// TwinCAT 3 PLC project Area2
// ProgramVersion: 3.1.4023.0
// libraries:
//   Tc2_DataExchange, * (Beckhoff Automation GmbH)
//   Tc2_MC2, * (Beckhoff Automation GmbH)
//   Tc2_Standard, * (Beckhoff Automation GmbH)
//   Tc2_System, * (Beckhoff Automation GmbH)
//   Tc2_TcpIp, * (Beckhoff Automation GmbH)
//   Tc2_Utilities, * (Beckhoff Automation GmbH)
//   Tc3_BA_Common, * (Beckhoff Automation GmbH)
//   Tc3_Database, * (Beckhoff Automation GmbH)
//   Tc3_JsonXml, * (Beckhoff Automation GmbH)
//   Tc3_Module, * (Beckhoff Automation GmbH)
// project tree:
//   COMMs_ADS/PROTOTYPE/ AdsClient_1.TcPOU (not stored), AdsHandle_1.TcPOU (not stored)
//   COMMs_ADS/Tasks/ AdsHandle.TcPOU, AdsClient.TcPOU (not stored)
//   COMMs_TCP/Types/ DUT.TcDUT (not stored), TcpData.TcDUT (not stored), TcpDataQueue.TcPOU
//   COMMs_TCP/Tasks/ TcpServer1Vision.TcPOU (not stored)
//   DUTs/Enums/ InsertionDirection.TcDUT (not stored), SectionEnum.TcDUT, Homing.TcDUT, SectionStatus.TcDUT, ConveyorMode.TcDUT (not stored), Cover.TcDUT (not stored), EventsEnum.TcTLEO (not stored), MaterialEnums.TcDUT (not stored), MaterialType.TcDUT (not stored), Surface.TcDUT
//   DUTs/Enums/Materials/ Cardboard.TcDUT (not stored), Chipboard.TcDUT (not stored), CornerGuard.TcDUT, WoodBunk.TcDUT (not stored)
//   DUTs/Enums/Robot Tasks/ A22.TcDUT, A21.TcDUT
//   DUTs/Hardware/ A21ToolStorage.TcDUT (not stored), FoldingMachine.TcDUT, Conveyor.TcPOU
//   DUTs/Hardware/Big Machines/ Robot.TcPOU, StrapMachine.TcPOU, WrapMachine.TcPOU
//   DUTs/Hardware/Insertion/Combinations/ ClampInsertion.TcPOU, PneumaticInsertion.TcPOU
//   DUTs/Hardware/Insertion/Drives/ AirPiston.TcPOU, ServoNC.TcPOU, TeknicEIP.TcPOU
//   DUTs/Hardware/Insertion/ Insertion.TcPOU, I_Insertion2D.TcIO
//   DUTs/Hardware/Material Storage/ MaterialStorage.TcPOU, WoodBunkTable.TcPOU
//   DUTs/ ONE_BIT.TcDUT, SuctionPad.TcDUT, VisionFrame.TcDUT (not stored), VisionSuite.TcDUT (not stored)
//   COMMs_ADS/Types/ AdsSocket.TcPOU (not stored), AdsDataQueue.TcPOU, AdsData.TcDUT (not stored)
//   DUTs/Bundle/ Bundle.TcDUT (not stored), CardboardMaterial.TcDUT (not stored), Interval.TcDUT (not stored), Material.TcDUT (not stored), PositionMaterials.TcDUT (not stored)
//   DUTs/Containers/ DynamicQueue.TcPOU, PtrQueue.TcPOU, IntQueue.TcPOU (not stored), Queue.TcPOU (not stored), StringQueue.TcPOU (not stored)
//   EventLogging/ EventLogger.TcIO (not stored), SqlDatabaseAccessor.TcPOU (not stored)
//   / GlobalTextList.TcGTLO (not stored), PlcTask.TcTTO (not stored)
//   GVLs/ GVL.TcGVL, Hardware.TcGVL, MultiProcess.TcGVL
//   POUs/ CallHardware.TcPOU, ConveyorControl.TcPOU, MAIN.TcPOU
//   POUs/Helper Functions/Document/ CreateJsonDocumentManual.TcPOU (not stored), CreateJsonDocumentAuto.TcPOU (not stored), FrameIsValid.TcPOU (not stored), VisionJsonParser.TcPOU
//   POUs/Helper Functions/General/ BufferIsEmpty.TcPOU (not stored), BundleIsValid.TcPOU (not stored), InRange.TcPOU (not stored), PositionIsValid.TcPOU (not stored), TimestructToString.TcPOU (not stored), WithinTolerance.TcPOU
//   POUs/Helper Functions/Material Functions/ GetPositionMasterLength.TcPOU, GetMaterialLength.TcPOU, MatchesMaterialType.TcPOU
//   POUs/Helper Functions/Misc/ ForceSetLifterConveyors.TcPOU, SizeCheck.TcPOU
//   Sections/Concrete/ AreaOutputEx.TcPOU, CardboardCornerGuardEx.TcPOU, ChipboardEx.TcPOU, PaperEx.TcPOU, WoodBunkEx.TcPOU
//   Sections/ I_MaterialSection.TcIO (not stored), SectionEx.TcPOU
// real-time tasks:
//   TASK PlcTask: cycle T#10ms, priority 20, ADS port 350

// ---- DUTs/Enums/Materials/CornerGuard.TcDUT
{attribute 'qualified_only'}
{attribute 'to_string'}
TYPE CornerGuard :
(
	COR48 := 1,
	COR96,
	
	size
);
END_TYPE

// ---- DUTs/Enums/Robot Tasks/A22.TcDUT
{attribute 'qualified_only'}
{attribute 'strict'}
TYPE A22 :
(
	IDLE,
	
	LOAD_CARDBOARD_TOP, //flat cardboards
	LOAD_CARDBOARD_BOTTOM,
	LOAD_CARDBOARD_SIDE,
	REMOVE_CARDBOARD_TOP,
	REMOVE_CARDBOARD_BOTTOM,
	REMOVE_CARDBOARD_SIDE,
	
	TRANSFER_TO_BENDER := 9, //corner cardboards
	TRANSFER_TO_OVERHEAD,
	REMOVE_CARDBOARD_FROM_BENDER,
	LOAD_BENDER_TO_UPPER_CORNER,
	LOAD_BENDER_TO_LOWER_CORNER,
	LOAD_OVERHEAD_TO_UPPER_CORNER,
	LOAD_OVERHEAD_TO_LOWER_CORNER,
	
	REMOVE_CARDBOARD_UPPER_CORNER,
	REMOVE_CARDBOARD_LOWER_CORNER,
	REMOVE_CARDBOARD_OVERHEAD := 18,
	
	LOAD_CORNER_GUARD_UPPER := 20, //corner guards
	LOAD_CORNER_GUARD_LOWER,
	REMOVE_CORNER_GUARD_UPPER,
	REMOVE_CORNER_GUARD_LOWER,
	
	size
);
END_TYPE

// ---- DUTs/Enums/SectionEnum.TcDUT
{attribute 'qualified_only'}
TYPE SectionEnum :
(
	NULL_SECTION := -1,
	PAPER,
	CARDBOARD_CORNERGUARD,
	CHIPBOARD,
	WOOD_BUNK,
	OUTPUT,
	
	size
);
END_TYPE

// ---- DUTs/Hardware/FoldingMachine.TcDUT
TYPE FoldingMachine :
STRUCT
	enable AT %Q* : BOOL;
	foldPos0 AT %Q* : REAL;
	foldPos1 AT %Q* : REAL;
	
	activeMaterial : STRING;
	
	ready AT %I* : BOOL;
	busy AT %I* : BOOL;
	done AT %I* : BOOL;
	error AT %I* : BOOL;
END_STRUCT
END_TYPE

// ---- DUTs/ONE_BIT.TcDUT
TYPE ONE_BIT :
STRUCT
	e1 : BIT;
END_STRUCT
END_TYPE

// ---- DUTs/Enums/Robot Tasks/A21.TcDUT
{attribute 'qualified_only'}
{attribute 'strict'}
TYPE A21 :
(
	IDLE,
	STAGE_BUNK,
	REMOVE_BUNK_FROM_STAGE,
	
	LOAD_BUNK_TO_TOP := 4,
	LOAD_BUNK_TO_SIDE,
	LOAD_BUNK_TO_BOTTOM,
	REMOVE_BUNK_FROM_TOP,
	REMOVE_BUNK_FROM_SIDE,
	REMOVE_BUNK_FROM_BOTTOM,
	
	GET_CHIPBOARD_FROM_SKID := 11,
	REMOVE_CHIPBOARD_FROM_TOOL,
	PLACE_CHIPBOARD_TO_TOP,
	PLACE_CHIPBOARD_TO_BOTTOM,
	REMOVE_CHIPBOARD_TOP,
	REMOVE_CHIPBOARD_BOTTOM,
	
	FIX_CHIPBOARD_ORIENTATION := 19,
	
	//testing only
	MOVE_HOME := 21,
	MOVE_POSITION1,
	MOVE_POSITION2,
	MOVE_UP,
	MOVE_DOWN,
	
	DIRECT_BUNK_TO_TOP := 27,
	DIRECT_BUNK_TO_SIDE,
	DIRECT_BUNK_TO_BOTTOM,
	
	INSPECT_BUNK := 31,
	INSPECT_CHIPBOARD,
	
	TOOL_CHANGE_BUNK := 34,
	TOOL_CHANGE_CHIPBOARD,
	
	size
);
END_TYPE

// ---- DUTs/Enums/Homing.TcDUT
{attribute 'qualified_only'}
{attribute 'strict'}
TYPE Homing :
(
	IDLE,
	HOME_OUT,
	HOME_FINAL,
	STOP,
	SET,
	DONE,
	REDO
);
END_TYPE

// ---- DUTs/Enums/SectionStatus.TcDUT
{attribute 'qualified_only'}
//{attribute 'strict'}
TYPE SectionStatus :
(
	IDLE,
	ALIGNING,
	ACTIVE,
	CLEARING,
	COMPLETE,
	
	size
);
END_TYPE

// ---- DUTs/Enums/Surface.TcDUT
{attribute 'qualified_only'}
//{attribute 'strict'}
TYPE Surface :
(
	TOP,
	LEFT,
	RIGHT,
	BOTTOM,
	
	TOP_LEFT,
	TOP_RIGHT,
	BOTTOM_LEFT,
	BOTTOM_RIGHT,
	
	size
);
END_TYPE

// ---- DUTs/SuctionPad.TcDUT
TYPE SuctionPad :
STRUCT
	enable AT %Q* : BOOL;
	readback AT %I* : BOOL;
END_STRUCT
END_TYPE

// ---- GVLs/GVL.TcGVL
{attribute 'qualified_only'}
VAR_GLOBAL CONSTANT
	maxPairs : USINT := 16;
	initArraySize : USINT := 4;
	maxQueue : INT := 16;
	
	nullPos : REAL := -1;
	
	numMaterials : INT := 32;
	allMaterials : ARRAY[0..numMaterials] OF Material := [
		(code := 'PAP28', width := 28, length := -1),
		
		(code := 'CAR20S', width := 20, length := 30),
		(code := 'CAR20M', width := 20, length := 45),
		(code := 'CAR20L', width := 20, length := 60),
		(code := 'CAR28S', width := 28, length := 30),
		(code := 'CAR28M', width := 28, length := 45),
		(code := 'CAR28L', width := 28, length := 60),
		
		(code := 'COR48', width := 1.5, length := 48),
		(code := 'COR96', width := 1.5, length := 96),
		
		(code := 'CIP18', width := 20, length := 18),
		(code := 'CIP54', width := 20, length := 54),
		
		(code := 'WDT20', width := 20, length := 2.5),
		(code := 'WDT22', width := 22, length := 2.5),
		(code := 'WDT28', width := 28, length := 2.5),
		
		(code := 'WDB20', width := 20, length := 2.5),
		(code := 'WDB22', width := 22, length := 2.5),
		(code := 'WDB28', width := 28, length := 2.5),
		
		(code := 'WDS08', width := 8, length := 2.5),
		(code := 'WDS10', width := 10, length := 2.5),
		(code := 'WDS12', width := 12, length := 2.5),
		(code := 'WDS14', width := 14, length := 2.5),
		(code := 'WDS8x8', width := 16, length := 2.5),
		(code := 'WDS8x10', width := 18, length := 2.5),
		(code := 'WDS20', width := 20, length := 2.5),
		(code := 'WDS22', width := 22, length := 2.5),
		(code := 'WDS12x12', width := 24, length := 2.5),
		(code := 'WDS12x14', width := 26, length := 2.5),
		(code := 'WDS28', width := 28, length := 2.5),
		(code := 'WDS20x10', width := 30, length := 2.5),
		(code := 'WDS20x12', width := 32, length := 2.5),
		
		(code := 'WDW20', width := 20, length := 6),
		(code := 'WDW22', width := 22, length := 6)]; //+1 null material

	nullBundle : Bundle;
	
	conveyorLength : REAL := 0;
	precisionTolerance : REAL := 0.05 * 25.4;
END_VAR
VAR_GLOBAL
	bundleOut : Bundle;
END_VAR

// ---- GVLs/Hardware.TcGVL
//{attribute 'qualified_only'}
VAR_GLOBAL CONSTANT
	numConveyors : INT := 20;
END_VAR
VAR_GLOBAL
	allConveyors : ARRAY[0..numConveyors] OF Conveyor;

	robots : ARRAY[1..6] OF Robot;
	
	(*
	names for moving parts should be in the following format: <type> <location> <left/right>
	*)
	
	//A23 - PAPER
	(*
	wrapperPaper : WrapMachine;
	*)
	//new
	wrapperA23 : WrapMachine;
	//-------------
	
	//A22 - CARDBOARD + CORNER GUARD
	(*
	cardboardSkid : ARRAY[Surface.LEFT..Surface.RIGHT] OF MaterialStorage;
	cornerGuardMagazine : ARRAY[Surface.LEFT..Surface.RIGHT] OF MaterialStorage;
	
	cardboardBender : ARRAY[Surface.LEFT..Surface.RIGHT] OF FoldingMachine;
	insertionCardboardCornerGuardSides : ARRAY[Surface.LEFT..Surface.RIGHT] OF ClampInsertion;
	insertionCardboardCornerGuardBottom : TeknicEIP;
	
	wrapperCardboardCornerguard : WrapMachine;
	*)
	//new
	cardboardBenderLeft, cardboardBenderRight : FoldingMachine;
	
	cardboardSkidLeft, cardboardSkidRight : MaterialStorage;
	cornerGuardMagazineLeft, cornerGuardMagazineRight : MaterialStorage;
	insertionA22Left, insertionA22Right : ClampInsertion;
	insertionA22Bottom : TeknicEIP;
	
	wrapperA22 : WrapMachine;
	overhead : STRING;
	//-------------
	
	
	//A21 - CHIPBOARD + WOOD BUNK
	(*
	toolStorage : ARRAY[Surface.LEFT..Surface.RIGHT] OF A21ToolStorage;
	
	chipboardSkid : ARRAY[Surface.LEFT..Surface.RIGHT] OF MaterialStorage;
	
	woodBunkMagazine : ARRAY[Surface.LEFT..Surface.RIGHT] OF MaterialStorage;
	stagingTable : ARRAY[Surface.LEFT..Surface.RIGHT] OF WoodBunkTable;
	strapper : StrapMachine;
	insertionWoodBunkSides : ARRAY[Surface.LEFT..Surface.RIGHT] OF PneumaticInsertion;
	insertionWoodBunkBottom : TeknicEIP;
	*)
	//new
	toolStorageA21Left, toolStorageA21Right : A21ToolStorage;
	
	chipboardSkidLeft, chipboardSkidRight : MaterialStorage;
	woodBunkMagazineLeft, woodBunkMagazineRight : MaterialStorage;
	
	stagingTableLeft, stagingTableRight : WoodBunkTable;
	strapperA21 : StrapMachine;
	
	insertionA21Left, insertionA21Right : PneumaticInsertion;	
	insertionA21Bottom : TeknicEIP;
	//-------------
	
	//A25 - OUTPUT
END_VAR

// ---- GVLs/MultiProcess.TcGVL
//{attribute 'qualified_only'}
VAR_GLOBAL
	iecCriticalSection : FB_IecCriticalSection; //must be used if communication routines are separated into their own core/task
END_VAR

// ---- DUTs/Hardware/Insertion/I_Insertion2D.TcIO
INTERFACE I_Insertion2D

METHOD ABSTRACT align : BOOL
VAR_INPUT
	targetPos : REAL;
END_VAR
END_METHOD

PROPERTY Busy : BOOL
GET
END_GET
SET
END_SET
END_PROPERTY

PROPERTY Contact : BOOL
GET
END_GET
SET
END_SET
END_PROPERTY

PROPERTY Home : BOOL
GET
END_GET
SET
END_SET
END_PROPERTY

METHOD ABSTRACT homingSequence : BOOL
VAR_INPUT
END_VAR
END_METHOD

METHOD ABSTRACT press : BOOL
VAR_INPUT
END_VAR
END_METHOD

METHOD ABSTRACT release : BOOL
VAR_INPUT
END_VAR
END_METHOD

PROPERTY ScrewPos : LREAL
GET
END_GET
SET
END_SET
END_PROPERTY

PROPERTY SliderPos : LREAL
GET
END_GET
SET
END_SET
END_PROPERTY

METHOD ABSTRACT traverse : BOOL
VAR_INPUT
	direction : MC_Direction;
END_VAR
END_METHOD

END_INTERFACE

// ---- DUTs/Hardware/Conveyor.TcPOU
FUNCTION_BLOCK Conveyor
VAR_OUTPUT
	operation : ConveyorMode;
	request : ConveyorMode;
	
	enable AT %Q* : BOOL := TRUE;
	direction AT %Q* : BOOL; //FALSE = forward, TRUE = backward
	pulse AT %Q* : BOOL;
	reset AT %Q* : BOOL;
	
	error AT %I* : BOOL;
	sensorEntry AT %I* : BOOL;
	sensorExit AT %I* : BOOL;
	
	//vertical conveyors only
	requestLifter: BOOL;

	lifterEnable AT %Q* : BOOL := TRUE;
	lifterDirection AT %Q* : BOOL; //FALSE = up, TRUE = down
	lifterPulse AT %Q* : BOOL;
	lifterReset AT %Q* : BOOL;
	
	lifterError AT %I* : BOOL;
	extended AT %I* : BOOL;
	retracted AT %I* : BOOL;
END_VAR
VAR_OUTPUT
	position AT %I* : REAL;
	velocity AT %I* : REAL;
END_VAR
VAR
	hasLifter : BOOL;
	
	//pulses are assumed to be low-high-low
	pulser : TP;
	lifterPulser : TP;
END_VAR
VAR_STAT CONSTANT
	pulseWidth : TIME := T#25MS;
END_VAR

pulser(IN:= , PT:= pulseWidth, Q=> pulse, ET=> );

direction := (operation = ConveyorMode.BACKWARD);

pulser.IN := 
	enable AND 
	NOT error AND 
	NOT reset AND 
	(operation = ConveyorMode.FORWARD OR operation = ConveyorMode.BACKWARD);

IF pulser.IN AND NOT pulser.Q THEN
	pulser.IN := FALSE;
END_IF

lifterPulser(IN:= , PT:= pulseWidth, Q=> lifterPulse, ET=> );

lifterPulser.IN := 
	hasLifter AND
	lifterEnable AND 
	NOT lifterError AND 
	NOT lifterReset AND 
	requestLifter;
	
IF lifterPulser.IN AND NOT lifterPulser.Q THEN
	lifterPulser.IN := FALSE;
END_IF

METHOD backward : BOOL
VAR_INPUT
END_VAR
END_METHOD

METHOD extend : BOOL
VAR_INPUT
END_VAR
END_METHOD

METHOD forward : BOOL
VAR_INPUT
END_VAR
END_METHOD

METHOD occupied : BOOL
occupied := sensorExit OR sensorEntry;
END_METHOD

METHOD reset : BOOL
VAR_INPUT
END_VAR
position := 0;
velocity := velocity; //no change

extend();
END_METHOD

METHOD retract : BOOL
VAR_INPUT
END_VAR
END_METHOD

METHOD setOperation : BOOL
VAR_INPUT
	newOperation : ConveyorMode;
END_VAR
operation := newOperation;
END_METHOD

METHOD setRequest : BOOL
VAR_INPUT
	requestedMode : ConveyorMode;
END_VAR
request := requestedMode;
END_METHOD

METHOD target : BOOL
VAR_INPUT
	targetPosition : REAL;
END_VAR
END_METHOD

END_FUNCTION_BLOCK

// ---- DUTs/Hardware/Big Machines/Robot.TcPOU
FUNCTION_BLOCK Robot
VAR_OUTPUT
	forceStop AT %Q* : BOOL;
	resetSignal AT %Q* : BOOL;
	
	taskID AT %Q* : INT;
	parameters AT %Q* : ARRAY[1..3] OF INT;
	
	outputs AT %Q* : ARRAY[1..50] OF INT;
	inputs AT %I* : ARRAY[1..20] OF INT;
	
	completedTask AT %I* : INT;
	tool AT %I* : SectionEnum;
	
	reserved : BOOL;
	reservation : SectionEnum := SectionEnum.NULL_SECTION;
	
	operational : BOOL;
	ready : BOOL;
	//busy : BOOL;
	done : BOOL;
	error : BOOL;
	errId : DINT;
END_VAR
VAR
	step : (SEND_COMMAND, WAIT);
END_VAR
VAR_STAT CONSTANT	
	emptyRegister : ARRAY[0..2] OF INT := [3(0)];
END_VAR

IF completedTask = taskID THEN
	done := TRUE;
END_IF

METHOD command : BOOL
VAR_INPUT
	task : INT;
	param1 : INT;
	param2 : INT;
	param3 : INT;
END_VAR
//command := reserve();

//IF command THEN
	(*
	taskId := task;
	parameters[1] := param1;
	parameters[2] := param2;
	parameters[3] := param3;
	*)
	
	outputs[1] := task;
	outputs[2] := param1;
	outputs[3] := param2;
	outputs[4] := param3;
//END_IF
END_METHOD

METHOD eStop : BOOL
VAR_INPUT
END_VAR
forceStop := TRUE;
eStop := TRUE;
END_METHOD

METHOD release : BOOL
VAR_INPUT
	sectionReservation : SectionEnum;
END_VAR
IF reservation = sectionReservation AND reserved THEN
	reservation := -1;
	reserved := FALSE;
	release := TRUE;
END_IF
END_METHOD

METHOD reserve : BOOL
VAR_INPUT
	sectionReservation : SectionEnum;
END_VAR
(*
some sections may use the same robot so it must be reserved before use
both sections need to check if the robot is open to commands before use
*)
IF
	(reserved AND reservation = SectionReservation) OR_ELSE
	(NOT reserved OR sectionReservation = SectionEnum.NULL_SECTION)
THEN
	reservation := sectionReservation;
	reserved := TRUE;
	reserve := TRUE;
END_IF
END_METHOD

METHOD reset : BOOL
release(reservation);

resetSignal := TRUE;
done := FALSE;
taskID := 0;
parameters := emptyRegister;

MEMSET(ADR(outputs), 0, SIZEOF(outputs));

IF ready AND completedTask = 0 THEN
	resetSignal := FALSE;
	reset := TRUE;
END_IF
END_METHOD

METHOD resume : BOOL
VAR_INPUT
END_VAR
forceStop := FALSE;

resume := NOT error AND errId = 0;
END_METHOD

METHOD setCommandAndWait : BOOL
VAR_INPUT
	task, param1, param2, param3 : INT;
END_VAR
(*
this method sends a command and waits for completion
MAKE SURE TO RESERVE THE ROBOT FIRST
*)
CASE step OF
	SEND_COMMAND: //send command
		command(
			task:= task, 
			param1:= param1, 
			param2:= param2, 
			param3:= param3);
		
		step := WAIT;
		
	WAIT:
		IF done THEN
			release(reservation);
			
			IF NOT reset() THEN
				RETURN;
			END_IF
			
			step := 0;
			
			setCommandAndWait := TRUE;
		END_IF
END_CASE
END_METHOD

METHOD setParamsAndWait : BOOL
VAR_INPUT
	newOutputs : REFERENCE TO ARRAY[1..50] OF INT;
END_VAR
outputs := newOutputs;

IF done THEN
	//release(); //let each section manually release
	
	IF NOT reset() THEN
		RETURN;
	END_IF
	
	step := 0;

	setParamsAndWait := TRUE;
END_IF
END_METHOD

END_FUNCTION_BLOCK

// ---- DUTs/Hardware/Big Machines/WrapMachine.TcPOU
FUNCTION_BLOCK WrapMachine
VAR_OUTPUT
	error AT %I* : BOOL;
	ready AT %I* : BOOL;
	busy AT %I* : BOOL;
	done (*AT %I**) : BOOL;
	home AT %I* : BOOL;
	
	rotations AT %Q* : INT;
	execute AT %Q* : BOOL;
	enable AT %Q* : BOOL;
	reset AT %Q* : BOOL;
	
	timeout : BOOL;
END_VAR
VAR
	holdPost : TON;
	delay : TON;
	
	start : BOOL;
	step : (SETUP, RUN, WAIT);
END_VAR
VAR_STAT CONSTANT
	pulseTime : TIME := T#100MS;
	holdTime : TIME := T#500MS;
	maxDelay : TIME := T#30S;
END_VAR

holdPost(IN:= , PT:= holdTime, Q=> , ET=> );
delay(IN:= step > 0, PT:= maxDelay, Q=> , ET=> );

IF delay.Q THEN
	delay.IN := FALSE;
	timeout := TRUE;
	busy := FALSE;
	step := SETUP;
END_IF

CASE step OF
	SETUP:
		busy := FALSE;
		IF error THEN
			reset := NOT reset;
			enable := FALSE;//NOT enable;
			
		ELSE
			reset := FALSE;
			enable := TRUE;
			
			IF start THEN
				start := FALSE;
				step := RUN;
			END_IF
			
		END_IF
	
	RUN:
		execute := TRUE;
		IF execute AND NOT home THEN
			execute := FALSE;
			step := WAIT;
		END_IF
		
	WAIT:
		IF home THEN
			holdPost.IN := TRUE;
			enable := FALSE;
			execute := FALSE;
		END_IF
		
		IF holdPost.Q THEN
			holdPost.IN := FALSE;
			done := TRUE;
			step := 0;
		END_IF
		
END_CASE

METHOD clear : BOOL
VAR_INPUT
END_VAR
(*
reset should be continuously called until machine returns evidence that it is ready again
machine is expected to not respond to reset signals if it is already in an idle state
*)
enable := FALSE;
execute := FALSE;

IF error THEN
	reset := NOT reset;
	clear := NOT error;

ELSE
	reset := FALSE;
	clear := TRUE;
	
END_IF
END_METHOD

METHOD wrap : BOOL
VAR_INPUT
	reqRotations : INT;
END_VAR
IF ready AND NOT busy AND NOT error THEN
	rotations := reqRotations;
	busy := TRUE;
	start := TRUE;
	wrap := TRUE;
END_IF
END_METHOD

END_FUNCTION_BLOCK

// ---- DUTs/Hardware/Material Storage/MaterialStorage.TcPOU
FUNCTION_BLOCK MaterialStorage
VAR_OUTPUT
	slots : ARRAY[1..GVL.maxQueue] OF STRING;
	//units : ARRAY[0..GVL.maxQueue] OF INT;
	
	empty AT %I* : ARRAY[1..GVL.maxQueue] OF BOOL;
END_VAR

METHOD findSlot : BOOL
VAR_INPUT
	materialID : STRING;
END_VAR
VAR_OUTPUT
	atSlot : INT := -1;
END_VAR
VAR
	i : INT;
END_VAR
IF materialID = '' THEN
	RETURN;
END_IF

FOR i:=0 TO GVL.maxQueue BY 1 DO
	IF slots[i] = materialID THEN
		atSlot := i;
		findSlot := TRUE;
		RETURN;
	END_IF
END_FOR
END_METHOD

METHOD getSlotsAsArray : POINTER TO STRING
getSlotsAsArray := ADR(slots);
END_METHOD

METHOD setupSlots : BOOL
VAR_INPUT
	setSlots : REFERENCE TO ARRAY[1..GVL.maxQueue] OF STRING;
END_VAR
slots := setSlots;
END_METHOD

END_FUNCTION_BLOCK

// ---- DUTs/Hardware/Insertion/Combinations/ClampInsertion.TcPOU
FUNCTION_BLOCK ClampInsertion EXTENDS Insertion
VAR
	slider : ServoNC;
	screw : TeknicEIP;
END_VAR

slider(
	bEnable:= enable, 
	home=> , 
	outerLimit=> , 
	innerLimit=> , 
	ready=> , 
	busy=> , 
	error=> , 
	homeSet=> , 
	position=> sliderPos);

screw(
	bEnable:= enable, 
	home=> , 
	outerLimit=> , 
	innerLimit=> , 
	done=> , 
	homeSet=> , 
	busy=> , 
	error=> , 
	position=> screwPos);

home := screw.home AND slider.home;
busy := slider.busy OR screw.busy;
error := slider.error OR screw.error;

METHOD align : BOOL
VAR_INPUT
	targetPos : REAL;
END_VAR
align := slider.moveAbsolute(targetPos := targetPos);
END_METHOD

METHOD homingSequence : BOOL
IF NOT slider.homeSet THEN
	slider.homingSequence();
END_IF

IF NOT screw.homeSet THEN
	screw.homingSequence();
END_IF

homingSequence := slider.homeSet AND screw.homeSet;
END_METHOD

METHOD press : BOOL
screw.moveContinuous(direction := MC_Negative_Direction);
END_METHOD

METHOD release : BOOL
VAR_INPUT
END_VAR
screw.moveContinuous(direction := MC_Positive_Direction);
END_METHOD

METHOD traverse : BOOL
VAR_INPUT
	direction : MC_Direction;
END_VAR
slider.moveContinuous(direction := direction);
END_METHOD

END_FUNCTION_BLOCK

// ---- DUTs/Hardware/Insertion/Insertion.TcPOU
FUNCTION_BLOCK ABSTRACT Insertion //IMPLEMENTS I_Insertion2D
VAR_INPUT CONSTANT
	enable : BOOL;
END_VAR
VAR_OUTPUT
	contact AT %I* : BOOL;
	home : BOOL;
	busy : BOOL;
	error : BOOL;
	
	sliderPos : LREAL;
	screwPos : LREAL;
END_VAR
(*
this abstract FB encapsulates 2 drives into a generic insertion machine
this FB cannot be used to instantiate insertions, it can only be used to refer/point to existing insertions
RETURN VALUES FOR THE METHODS ARE MEANINGLESS
*)

METHOD ABSTRACT align : BOOL
VAR_INPUT
	targetPos : REAL;
END_VAR
END_METHOD

METHOD ABSTRACT homingSequence : BOOL
VAR_INPUT
END_VAR
END_METHOD

METHOD ABSTRACT press : BOOL
VAR_INPUT
END_VAR
END_METHOD

METHOD ABSTRACT release : BOOL
VAR_INPUT
END_VAR
END_METHOD

METHOD ABSTRACT traverse : BOOL
VAR_INPUT
	direction : MC_Direction;
END_VAR
END_METHOD

END_FUNCTION_BLOCK

// ---- DUTs/Hardware/Insertion/Drives/ServoNC.TcPOU
FUNCTION_BLOCK ServoNC
VAR_INPUT CONSTANT
	bEnable : BOOL;
END_VAR
VAR_OUTPUT
	home AT %I* : BOOL;
	outerLimit AT %I* : BOOL;
	innerLimit AT %I* : BOOL;
	
	ready : BOOL;
	busy : BOOL;
	error : BOOL;
	homeSet : BOOL;
	
	position : LREAL;
END_VAR
VAR
	axis : AXIS_REF;
	
	mcReadPosition : MC_ReadActualPosition;
	mcReset : MC_Reset;
	
	mcPower : MC_Power;
	mcMoveAbsolute : MC_MoveAbsolute;
	mcMoveRelative : MC_MoveRelative;
	mcMoveVelocity : MC_MoveVelocity;
	
	mcStop : MC_Stop;
	mcSetPosition : MC_SetPosition;
	
	step : Homing;
END_VAR
VAR_STAT CONSTANT
	targetingVelocity : INT := 500;
	continuousVelocity : INT := 200;
END_VAR

mcReadPosition(
	Axis:= axis, 
	Enable:= TRUE, 
	Valid=> , 
	Busy=> , 
	Error=> , 
	ErrorID=> , 
	Position=> position);

mcReset(
	Axis:= axis, 
	Execute:= , 
	Done=> , 
	Busy=> , 
	Error=> , 
	ErrorID=> );

mcPower(
	Axis:= axis, 
	Enable:= bEnable, 
	Enable_Positive:= TRUE, 
	Enable_Negative:= TRUE, 
	Override:= 100, 
	BufferMode:= , 
	Options:= , 
	Status=> , 
	Busy=> , 
	Active=> , 
	Error=> , 
	ErrorID=> );

mcMoveAbsolute(
	Axis:= axis, 
	Execute:= , 
	Position:= , 
	Velocity:= targetingVelocity, 
	Acceleration:= , 
	Deceleration:= , 
	Jerk:= , 
	BufferMode:= , 
	Options:= , 
	Done=> , 
	Busy=> , 
	Active=> , 
	CommandAborted=> , 
	Error=> , 
	ErrorID=> );
		
mcMoveRelative(
	Axis:= axis, 
	Execute:= , 
	Distance:= ,
	Velocity:= targetingVelocity, 
	Acceleration:= , 
	Deceleration:= , 
	Jerk:= , 
	BufferMode:= , 
	Options:= , 
	Done=> , 
	Busy=> , 
	Active=> , 
	CommandAborted=> , 
	Error=> , 
	ErrorID=> );
	
mcMoveVelocity(
	Axis:= axis, 
	Execute:= , 
	Velocity:= continuousVelocity, 
	Acceleration:= , 
	Deceleration:= , 
	Jerk:= , 
	Direction:= , 
	BufferMode:= , 
	Options:= , 
	InVelocity=> , 
	Busy=> , 
	Active=> , 
	CommandAborted=> , 
	Error=> , 
	ErrorID=> );
	
mcStop(
	Axis:= axis, 
	Execute:= , 
	Deceleration:= , 
	Jerk:= , 
	Options:= , 
	Done=> , 
	Busy=> , 
	Active=> , 
	CommandAborted=> , 
	Error=> , 
	ErrorID=> );

mcSetPosition(
	Axis:= axis, 
	Execute:= , 
	Position:= , 
	Mode:= , 
	Options:= , 
	Done=> , 
	Busy=> , 
	Error=> , 
	ErrorID=> );
	
busy := mcMoveAbsolute.Busy OR mcMoveRelative.Busy OR mcMoveVelocity.Busy OR mcSetPosition.Busy OR mcReset.Busy OR mcStop.Busy OR step <> 0;
error := mcMoveAbsolute.Error OR mcMoveRelative.Error OR mcMoveVelocity.Error OR mcSetPosition.Error OR mcReset.Error OR mcStop.Error OR step <> 0;
ready := bEnable AND NOT busy AND homeSet;

IF step <> 0 THEN
	mcReset.Execute := FALSE;
	mcMoveAbsolute.Execute := FALSE;
	mcMoveRelative.Execute := FALSE;
	mcMoveVelocity.Execute := FALSE;
	mcStop.Execute := FALSE;
	mcSetPosition.Execute := FALSE;
END_IF

METHOD homingSequence : BOOL
CASE step OF
	Homing.IDLE:
		IF bEnable THEN
			step := Homing.REDO;
		END_IF
		
	Homing.REDO:
		IF mcMoveVelocity.Execute AND NOT innerLimit THEN
			mcMoveVelocity.Execute := FALSE;
			step := Homing.HOME_OUT;
			RETURN;
		END_IF
		
		mcMoveVelocity.Direction := MC_Negative_Direction;
		mcMoveVelocity.Execute := TRUE;
		
	Homing.HOME_OUT:
		IF mcMoveVelocity.Execute AND NOT home THEN //if reached home
			mcMoveVelocity.Execute := FALSE;
			step := Homing.STOP;
			RETURN;
		END_IF
		
		mcMoveVelocity.Direction := MC_Positive_Direction;
		mcMoveVelocity.Execute := TRUE;
		
	Homing.STOP:
		IF mcStop.Execute AND mcStop.Done THEN
			mcStop.Execute := FALSE;
			step := Homing.SET;
			RETURN;
		END_IF
		
		mcStop.Execute := TRUE;
		
	Homing.SET:
		IF mcSetPosition.Execute AND mcSetPosition.Done THEN
			mcSetPosition.Execute := FALSE;
			homingSequence := TRUE;
			step := Homing.IDLE;
			RETURN;
		END_IF
		
		mcSetPosition.Position := 0;
		mcSetPosition.Execute := TRUE;
		
END_CASE
END_METHOD

METHOD moveAbsolute : BOOL
VAR_INPUT
	targetPos : LREAL;
END_VAR
IF NOT busy AND NOT error THEN
	mcMoveAbsolute.Position := targetPos;
END_IF
moveAbsolute := mcMoveAbsolute.Done;
END_METHOD

METHOD moveContinuous : BOOL
VAR_INPUT
	direction : MC_Direction;
END_VAR
mcMoveVelocity.Direction := direction;

mcMoveVelocity.Execute := TRUE;

moveContinuous := NOT mcMoveVelocity.Error;
END_METHOD

METHOD moveRelative : BOOL
VAR_INPUT
	distance : LREAL;
END_VAR
mcMoveRelative.Distance := distance;

moveRelative := mcMoveRelative.Done;
END_METHOD

METHOD reset : BOOL
VAR_INPUT
END_VAR
mcReset.Execute := TRUE;

reset := mcReset.Done;
END_METHOD

METHOD stop : BOOL
VAR_INPUT
END_VAR
END_METHOD

END_FUNCTION_BLOCK

// ---- DUTs/Hardware/Insertion/Drives/TeknicEIP.TcPOU
FUNCTION_BLOCK TeknicEIP //EXTENDS EncodedDrive
VAR_INPUT CONSTANT
	bEnable : BOOL;
END_VAR
VAR_OUTPUT
	enable AT %Q* : BOOL; //enable + pulses
	A AT %Q* : BOOL; //direction (F = inwards, T = outwards)
	B AT %Q* : BOOL; //home bit
	brakeRelease AT %Q* : BOOL;
	
	contact AT %I* : BOOL;
	
	home AT %I* : BOOL;
	outerLimit AT %I* : BOOL;
	innerLimit AT %I* : BOOL;
	done AT %I* : BOOL;	
	
	homeSet : BOOL;
	busy : BOOL;
	error : BOOL;
	
	position : LREAL;
	targetPos : LREAL;
END_VAR
VAR
	mode : (HOLD, TARGET, CONTINUOUS);
	
	resetTimer : TP;
	pulser : TON;
	requestedPulses : INT;
	
	step : Homing;//(IDLE, HOME_UP, HOME_FINAL, DOWN, REDO_HOME, HOME_DONE);
END_VAR
VAR_STAT CONSTANT
	resetTime : TIME := T#1000MS;
	pulseWidth : TIME := T#25MS;
	unitsPerPulse : INT := 800; //800 Teknic units per revolution
	distancePerPulse : INT := 5; //5mm per revolution
END_VAR

IF NOT bEnable THEN
	RETURN;
END_IF

resetTimer(IN:= , PT:= resetTime, Q=> , ET=> );
IF resetTimer.Q THEN
	brakeRelease := FALSE;
	enable := FALSE;
	RETURN;
END_IF
resetTimer.IN := FALSE;


CASE mode OF
	HOLD:
		//
	
	TARGET:
		IF WithinTolerance(position, target, unitsPerPulse) THEN
			requestedPulses := 0;
			mode := HOLD;
			
		ELSIF position < target THEN
			A := TRUE;
			requestPulses(1);
		ELSIF position > target THEN
			A := FALSE;
			requestPulses(1);
		END_IF

	CONTINUOUS:
		requestPulses(1);
		
END_CASE

IF home OR innerLimit OR outerLimit THEN
	requestedPulses := 0;
	mode := HOLD;
END_IF

sequence();

METHOD homingSequence : BOOL
CASE step OF
	Homing.IDLE:
		enable := FALSE;
		A := FALSE;
		B := FALSE;
		brakeRelease := TRUE;
		
		homeSet := FALSE;
		step := Homing.REDO;
		
	Homing.REDO: //let insertion drop to inner limit before homing
		enable := FALSE;
		A := FALSE;
		B := FALSE;
		brakeRelease := TRUE;
		
		IF NOT innerLimit THEN
			enable := TRUE;
			step := Homing.HOME_OUT;
		END_IF
	
	Homing.HOME_OUT:
		enable := TRUE;
		A := FALSE;
		B := TRUE;
		brakeRelease := TRUE;
		
		IF NOT home THEN
			B := FALSE;
			step := Homing.DONE;
		END_IF
		
	Homing.DONE:
		enable := TRUE;
		A := FALSE;
		B := FALSE;
		brakeRelease := TRUE;
		
		position := 0;
		homeSet := TRUE;
		homingSequence := TRUE;
		step := Homing.IDLE;
	
END_CASE
END_METHOD

METHOD moveAbsolute : BOOL
VAR_INPUT
	targetPos : LREAL;
END_VAR
targetPos := target;
mode := TARGET;
END_METHOD

METHOD moveContinuous : BOOL
VAR_INPUT
	direction : MC_Direction;
END_VAR
IF direction = MC_Negative_Direction THEN
	A := FALSE;
ELSIF direction = MC_Positive_Direction THEN
	A := TRUE;
END_IF

mode := CONTINUOUS;
END_METHOD

METHOD PRIVATE requestPulses : BOOL
VAR_INPUT
	request : INT;
END_VAR
IF (done OR requestedPulses = 0) AND request > 0 THEN
	requestedPulses := request;
	
	requestPulses := TRUE;
END_IF
END_METHOD

METHOD reset : BOOL
VAR_INPUT
END_VAR
resetTimer.IN := TRUE;
END_METHOD

METHOD sequence : BOOL
VAR_INPUT
END_VAR
pulser(IN:= , PT:= pulseWidth, Q=> , ET=> ); //when timer is enabled, this toggles enable every <pulseWidth>

IF requestedPulses = 0 THEN
	busy := FALSE;
	
	enable := TRUE;
	pulser.IN := FALSE;
	RETURN;
END_IF

busy := TRUE;
pulser.IN := TRUE;

IF pulser.Q THEN
	pulser.IN := FALSE;
	enable := NOT enable;
	
	IF enable THEN //enable is TRUE after toggle
		requestedPulses := requestedPulses - 1;
		
		IF A THEN
			position := position + distancePerPulse;
		ELSE
			position := position - distancePerPulse;
		END_IF
	END_IF
	
END_IF
END_METHOD

END_FUNCTION_BLOCK

// ---- POUs/Helper Functions/General/WithinTolerance.TcPOU
FUNCTION WithinTolerance : BOOL
VAR_INPUT
	v1 : LREAL;
	v2 : LREAL;
	tolerance : LREAL;
END_VAR

WithinTolerance := ABS(v1-v2) < tolerance;

END_FUNCTION

// ---- DUTs/Hardware/Material Storage/WoodBunkTable.TcPOU
FUNCTION_BLOCK WoodBunkTable EXTENDS MaterialStorage
VAR
	//slots : ARRAY[1..numSlots] OF STRING;
	occupied AT %I* : ARRAY[1..numSlots] OF BOOL;
	//sensors must turn HIGH before bunk arrives, and turn LOW after bunk leaves
	
	i : INT(1..10);
END_VAR
VAR_STAT CONSTANT
	numSlots : INT := 10;
END_VAR

FOR i:=1 TO numSlots BY 1 DO
	IF NOT occupied[i] THEN
		slots[i] := '';
	END_IF
END_FOR

METHOD autofill : BOOL
VAR_INPUT
	materialID : STRING;
END_VAR
VAR
	i : INT;
	slot : INT;
END_VAR
(*
this method will automatically find an open slot
*)
IF isFull() OR materialID = '' THEN
	RETURN;
END_IF

IF findOpenSlot(materialID, openSlot=> slot) THEN
	place(slot, materialID);
	autofill := TRUE;
END_IF
END_METHOD

METHOD findOpenSlot : BOOL
VAR_INPUT
	materialID : STRING;
END_VAR
VAR_OUTPUT
	openSlot : INT := 0;
END_VAR
VAR
	i : INT;
END_VAR
IF FIND(materialID, 'WDW') > 0 THEN //top wide, load in slot 0-1
	FOR i:=1 TO 2 BY 1 DO
		IF NOT occupied[i] THEN
			findOpenSlot := TRUE;
			openSlot := i;
			RETURN;
		END_IF
	END_FOR
	
ELSIF FIND(materialID, 'WDT') > 0 OR FIND(materialID, 'WDS') > 0 THEN //top std and sides, load in slot 2-9
	FOR i:=3 TO 10 BY 1 DO
		IF NOT occupied[i] THEN
			findOpenSlot := TRUE;
			openSlot := i;
			RETURN;
		END_IF
	END_FOR
	
END_IF
END_METHOD

METHOD findSlot : BOOL
VAR_INPUT
	materialID : STRING;
END_VAR
VAR_OUTPUT
	atSlot : INT;
END_VAR
VAR
	i : INT;
END_VAR
FOR i:=1 TO numSlots BY 1 DO
	IF slots[i] = materialID THEN
		atSlot := i;
		findSlot := TRUE;
		RETURN;
	END_IF
END_FOR
END_METHOD

METHOD isEmpty : BOOL
VAR
	i : INT;
	temp : BOOL;
END_VAR
FOR i:=1 TO numSlots BY 1 DO
	temp := temp OR occupied[i]; //TRUE if any slots are occupied
END_FOR

isEmpty := NOT temp; //invert result - FALSE if any slots are occupied
END_METHOD

METHOD isFull : BOOL
VAR
	i : INT;
	temp : BOOL := TRUE;
END_VAR
FOR i:=1 TO numSlots BY 1 DO
	temp := temp AND occupied[i];
END_FOR

isFull := TEMP;
END_METHOD

METHOD place : BOOL
VAR_INPUT
	i : INT;
	materialID : STRING;
END_VAR
IF slots[i] = '' AND NOT occupied[i] THEN
	slots[i] := materialID;
	place := TRUE;
END_IF
END_METHOD

METHOD remove : BOOL
VAR_INPUT
	i : INT;
END_VAR
VAR_OUTPUT
	materialID : STRING;
END_VAR
IF slots[i] <> '' AND occupied[i] THEN
	materialID := slots[i];
	slots[i] := '';
	
	remove := TRUE;
END_IF
END_METHOD

END_FUNCTION_BLOCK

// ---- DUTs/Hardware/Big Machines/StrapMachine.TcPOU
FUNCTION_BLOCK StrapMachine
VAR_OUTPUT
	error AT %I* : BOOL;
	ready AT %I* : BOOL;
	busy AT %I* : BOOL;
	done (*AT %I**) : BOOL;
	home AT %I* : BOOL;
	
	execute AT %Q* : BOOL;
	enable AT %Q* : BOOL;
	reset AT %Q* : BOOL;
	
	timeout : BOOL;
END_VAR
VAR
	topSuction AT %Q* : BOOL;
	bottomSuction AT %Q* : BOOL;
	
	holdPost : TON;
	delay : TON;
	
	start : BOOL;
	step : (SETUP, RUN, WAIT);
END_VAR
VAR_STAT CONSTANT
	pulseTime : TIME := T#100MS;
	holdTime : TIME := T#500MS;
	maxDelay : TIME := T#30S;
END_VAR

holdPost(IN:= , PT:= holdTime, Q=> , ET=> );
delay(IN:= step > 0, PT:= maxDelay, Q=> , ET=> );

IF delay.Q THEN
	delay.IN := FALSE;
	timeout := TRUE;
	busy := FALSE;
	step := SETUP;
END_IF

CASE step OF
	SETUP:
		busy := FALSE;
		IF error THEN
			reset := NOT reset;
			enable := FALSE;//NOT enable;
			
		ELSE
			reset := FALSE;
			enable := TRUE;
			
			IF start THEN
				start := FALSE;
				step := RUN;
			END_IF
			
		END_IF
	
	RUN:
		execute := TRUE;
		IF execute AND NOT home THEN
			execute := FALSE;
			step := WAIT;
		END_IF
		
	WAIT:
		IF home THEN
			holdPost.IN := TRUE;
			enable := FALSE;
			execute := FALSE;
		END_IF
		
		IF holdPost.Q THEN
			holdPost.IN := FALSE;
			done := TRUE;
			step := 0;
		END_IF
		
END_CASE

(*
executePulse(IN:= , PT:= pulseTime, Q=> , ET=> );
execute := executePulse.IN AND NOT executePulse.Q;

IF executePulse.Q THEN
	executePulse.IN := FALSE;
END_IF


resetPulse(IN:= , PT:= pulseTime, Q=> , ET=> );
StrapMachineST.reset := resetPulse.IN AND NOT resetPulse.Q;

IF resetPulse.Q THEN
	executePulse.IN := FALSE;
END_IF

ready := enable AND NOT execute AND NOT StrapMachineST.reset AND NOT error AND home;
*)

METHOD clear : BOOL
VAR_INPUT
END_VAR
(*
reset should be continuously called until machine returns evidence that it is ready again
machine is expected to not respond to reset signals if it is already in an idle state
*)
enable := FALSE;
execute := FALSE;

IF error THEN
	reset := NOT reset;
	clear := NOT error;

ELSE
	reset := FALSE;
	clear := TRUE;
	
END_IF
END_METHOD

METHOD strap : BOOL
VAR_INPUT
END_VAR
IF ready AND NOT busy AND NOT error THEN
	busy := TRUE;
	start := TRUE;
	strap := TRUE;
END_IF
END_METHOD

END_FUNCTION_BLOCK

// ---- DUTs/Hardware/Insertion/Combinations/PneumaticInsertion.TcPOU
FUNCTION_BLOCK PneumaticInsertion EXTENDS Insertion
VAR
	slider : TeknicEIP;
	screw : AirPiston;
END_VAR

slider(
	bEnable:= enable, 
	home=> , 
	outerLimit=> , 
	innerLimit=> , 
	done=> , 
	homeSet=> , 
	busy=> , 
	error=> , 
	position=> sliderPos);
	
screw(
	bEnable:= enable, 
	direction=> , 
	valveIn=> , 
	valveOut=> , 
	contact=> , 
	home=> , 
	innerLimit=> , 
	ready=> , 
	busy=> , 
	error=> , 
	homeSet=> );
	
home := screw.home AND slider.home;
busy := slider.busy OR screw.busy;
error := slider.error OR screw.error;

METHOD align : BOOL
VAR_INPUT
	targetPos : REAL;
END_VAR
align := slider.moveAbsolute(targetPos := targetPos);
END_METHOD

METHOD homingSequence : BOOL
IF NOT screw.homeSet THEN
	screw.homingSequence();
END_IF

IF NOT slider.homeSet THEN
	slider.homingSequence();
END_IF

homingSequence := screw.homeSet AND slider.homeSet;
END_METHOD

METHOD press : BOOL
screw.slideIn();
END_METHOD

METHOD release : BOOL
VAR_INPUT
END_VAR
screw.slideOut();
END_METHOD

METHOD traverse : BOOL
VAR_INPUT
	direction : MC_Direction;
END_VAR
slider.moveContinuous(direction := direction);
END_METHOD

END_FUNCTION_BLOCK

// ---- DUTs/Hardware/Insertion/Drives/AirPiston.TcPOU
FUNCTION_BLOCK AirPiston
VAR_IN_OUT CONSTANT
	bEnable : BOOL;
END_VAR
VAR_OUTPUT	
	valveIn AT %Q* : BOOL;
	valveOut AT %Q* : BOOL;
	
	contact AT %I* : BOOL;
	
	home AT %I* : BOOL;
	innerLimit AT %I* : BOOL;
	
	ready : BOOL;
	busy : BOOL;
	error : BOOL;
	homeSet : BOOL;
END_VAR
VAR
	direction : (IN, OUT, HOLD);
	step : Homing;
END_VAR

IF NOT bEnable THEN
	valveIn := FALSE;
	valveOut := FALSE;
	RETURN;
END_IF

IF home OR innerLimit (*OR outerLimit*) THEN
	direction := HOLD;
END_IF

CASE direction OF
	HOLD:
		valveIn := FALSE;
		valveOut := FALSE;
		
	IN:
		valveIn := TRUE;
		valveOut := FALSE;
		
	OUT:
		valveIn := FALSE;
		valveOut := TRUE;
		
END_CASE

METHOD homingSequence : BOOL
(*
this version of homing always traverses to the inner limit before returning to home,
eliminating the possibility of reaching the outer limit while homing
*)
CASE step OF
	Homing.IDLE:
		step := Homing.REDO;
		
	Homing.REDO: //technically HOME_IN, towards travel limit
		valveIn := TRUE;
		valveOut := FALSE;
		
		IF NOT innerLimit THEN
			valveIn := FALSE;
			valveOut := FALSE;
			step := Homing.HOME_OUT;
		END_IF
		
	Homing.HOME_OUT: //towards home
		valveIn := FALSE;
		valveOut := TRUE;
		
		IF NOT home THEN //if reached home
			valveIn := FALSE;
			valveOut := FALSE;
			step := Homing.DONE;
		END_IF
		
	Homing.DONE:
		valveIn := FALSE;
		valveOut := FALSE;
		homeSet := TRUE;
		
		homingSequence := TRUE;		
	
END_CASE
END_METHOD

METHOD slideIn : BOOL
VAR_INPUT
END_VAR
direction := IN;

slideIn := TRUE;
END_METHOD

METHOD slideOut : BOOL
VAR_INPUT
END_VAR
direction := OUT;

slideOut := TRUE;
END_METHOD

METHOD stop : BOOL
VAR_INPUT
END_VAR
valveIn := FALSE;
valveOut := FALSE;
direction := HOLD;

stop := TRUE;
END_METHOD

END_FUNCTION_BLOCK

// ---- COMMs_ADS/Tasks/AdsHandle.TcPOU
FUNCTION_BLOCK AdsHandle
VAR_INPUT
	ServerNetId			: STRING; 	(* Server AmsNetId *)
	ServerPort 			: UDINT;	(* Server port number *)
	
	remoteAccessPrefix	: STRING;
END_VAR
VAR_OUTPUT
	bBusy				: BOOL;
	err					: BOOL;
	errid				: UDINT;
	
	receiveBuffer		: ARRAY[0..100000] OF BYTE; //TCP style data buffer
	receiveStruct		: AdsData;
END_VAR
VAR	
	socket 				: AdsSocket; //only this needs initialization
	
	sendQueue			: AdsDataQueue;
	sendBufferQueue 	: DynamicQueue; //anything going into this needs to be a TcpStruct
	
	sendBuffer 			: ARRAY[0..50000] OF BYTE; //temp byte buffer to send if neccessary
	sendStruct			: AdsData;
	
	//setupStep 			: (CLOSE_CONNECTIONS, CREATE_LISTENER, ACCEPT_CONNECTION, FINISH_SETUP);
	sendDelay : TON;
END_VAR
VAR_STAT CONSTANT
	emptyData : AdsData;
	sendDelayTime : TIME := T#1S;
END_VAR

sendDelay(IN:= , PT:= sendDelayTime, Q=> , ET=> );
sendDelay.IN := TRUE;

IF sendDelay.Q THEN
	
	sendStruct := sendQueue.poll();
	IF MEMCMP(ADR(sendStruct), ADR(emptyData), SIZEOF(AdsData)) <> 0 THEN //if valid data to send
	
		write(
			symbol := CONCAT(remoteAccessPrefix, 'receiveStruct'),
			data := ADR(sendStruct),
			dataSize := SIZEOF(sendStruct));
			
		sendDelay.IN := FALSE;
	END_IF
	
END_IF

METHOD clearBuffer : BOOL
VAR
	emptyReceiverStruct : AdsData;
END_VAR
//MEMSET(ADR(receiveBuffer), 0, SIZEOF(receiveBuffer));
receiveStruct := emptyReceiverStruct;
END_METHOD

METHOD close : BOOL
VAR_INPUT
END_VAR
socket.close();
END_METHOD

METHOD getHandlerName : STRING
getHandlerName := socket.remotePrgName;
END_METHOD

METHOD open : BOOL
VAR_INPUT
	localPrgName : STRING;
	localNetId : T_AmsNetId;
	localPort : T_AmsPort;
END_VAR
socket.open(localPrgName, localNetId, localPort);
END_METHOD

METHOD queueData : BOOL
VAR_INPUT
	data : REFERENCE TO AdsData;
END_VAR
//MEMCPY(ADR(temp), data.pValue, data.diSize);
sendQueue.push(data);
END_METHOD

METHOD read : BOOL
VAR_INPUT
	symbol : STRING;
	buffer : PVOID;
	symbolSize : UDINT;
END_VAR
IF NOT socket.readBusy THEN
	read := socket.read(
		symbol:= symbol,
		buffer := buffer,
		symbolSize := symbolSize);
END_IF
END_METHOD

METHOD write : BOOL
VAR_INPUT
	symbol : STRING;
	data : PVOID;
	dataSize : UDINT;
END_VAR
VAR
	timer : TON;
END_VAR
IF NOT socket.writeBusy THEN
	write := socket.write(
		symbol:= symbol,
		data := data,
		dataSize := dataSize);
END_IF
END_METHOD

END_FUNCTION_BLOCK

// ---- COMMs_ADS/Types/AdsDataQueue.TcPOU
{attribute 'call_after_init'}
FUNCTION_BLOCK AdsDataQueue
VAR
	elements : FB_BA_DynamicArray := (uiEntrySize := SIZEOF(POINTER TO AdsData), uiMinExpCount := GVL.initArraySize); 
	length : INT := 0;
	
	entrySize : UDINT;
END_VAR
(*
this container stores dynamically generated AdsData Structs
AdsData to be added are passed by reference, then this function block allocates a structure to be stored
AdsData are get() by reference and poll() by value
*)

METHOD clear : BOOL
VAR
	i : INT;
	temp : REFERENCE TO AdsData;
	tempAdr : POINTER TO AdsData;
END_VAR
FOR i:=0 TO length-1 BY 1 DO
	temp := get(index := i, getSize => );
	tempAdr := ADR(temp);
	__DELETE(tempAdr);
END_FOR

elements.Reset();
length := 0;
END_METHOD

METHOD contains : BOOL //check contents, not pointer value
VAR_INPUT
	value : REFERENCE TO AdsData;
END_VAR
VAR_OUTPUT
	atIndex : INT;
END_VAR
VAR
	temp : REFERENCE TO AdsData;
	i : INT;
END_VAR
IF length = 0 THEN
	contains := FALSE;
	RETURN;
END_IF

FOR i:=0 TO length-1 BY 1 DO
	temp := get(index := i, getSize => );
	
	IF 
		SIZEOF(value) = entrySize AND //same size
		MEMCMP(ADR(temp), ADR(value), SIZEOF(entrySize)) = 0 //same data
	THEN
		contains := TRUE;
		atIndex := i;
		RETURN;
	END_IF
	
END_FOR
contains := FALSE;
END_METHOD

METHOD get : REFERENCE TO AdsData
VAR_INPUT
	index : INT;
END_VAR
VAR_OUTPUT
	getSize : UDINT;
END_VAR
IF length = 0 OR index < 0 OR index >= length THEN
	getSize := 0;
ELSE
	elements.GetEntry(diIndex := index, pResultEntry := ADR(get));
	getSize := SIZEOF(get);
END_IF
END_METHOD

METHOD isEmpty : BOOL
VAR_INPUT
END_VAR
isEmpty := length = 0;
END_METHOD

METHOD poll : AdsData
VAR_OUTPUT
	getSize : UDINT;
END_VAR
IF length > 0 THEN
	poll := get(index := 0, getSize => getSize);
	elements.RemoveEntry(diIndex := 0);
	
	length := length - 1;
END_IF
END_METHOD

METHOD push : BOOL
VAR_INPUT
	value : REFERENCE TO AdsData;
END_VAR
VAR
	temp : POINTER TO AdsData;
END_VAR
temp := __NEW(AdsData);
temp^ := value;

elements.AddEntryPtr(pEntry := temp);

length := length + 1;
END_METHOD

METHOD set : BOOL
VAR_INPUT
	i : INT;
	value : REFERENCE TO AdsData;
END_VAR
VAR
	temp : REFERENCE TO AdsData;
END_VAR
IF length = 0 THEN
	RETURN;
END_IF

IF i >= 0 AND i < length THEN
	temp REF= get(i);
	temp := value;
	
	set := TRUE;
END_IF
END_METHOD

{attribute 'call_after_init'}
METHOD setup : BOOL
VAR_INPUT
END_VAR
entrySize := SIZEOF(AdsData);
END_METHOD

METHOD size : INT
size := length;
END_METHOD

END_FUNCTION_BLOCK

// ---- DUTs/Containers/DynamicQueue.TcPOU
FUNCTION_BLOCK DynamicQueue
VAR
	elements : FB_BA_DynamicArray := (uiEntrySize := SIZEOF(POINTER TO BYTE), uiMinExpCount := GVL.initArraySize); 
	elementSizes : FB_BA_DynamicArray := (uiEntrySize := SIZEOF(LINT), uiMinExpCount := GVL.initArraySize);
	length : INT := 0;
END_VAR
(*
this dynamic array stores pointers to dynamically generated objects
elements to be added are passed by value, then this function block allocates bytes
*)

METHOD clear : BOOL
VAR
	i : INT;
	temp : POINTER TO BYTE;
END_VAR
FOR i:=0 TO length-1 BY 1 DO
	temp := get(index := i);
	__DELETE(temp);
END_FOR


elements.Reset();
elementSizes.Reset();
length := 0;
END_METHOD

METHOD contains : BOOL
VAR_INPUT
	value : ANY;
END_VAR
VAR_OUTPUT
	atIndex : INT;
END_VAR
VAR
	temp : POINTER TO BYTE;
	tempSize : LINT;
	i : INT;
END_VAR
IF length = 0 THEN
	contains := FALSE;
	RETURN;
END_IF

FOR i:=0 TO length-1 BY 1 DO
	temp := get(index := i, getSize => tempSize);
	
	IF 
		tempSize = value.diSize AND //same size
		MEMCMP(get(i), value.pValue, TO_UDINT(value.diSize)) = 0 //same data
	THEN
		contains := TRUE;
		atIndex := i;
		RETURN;
	END_IF
	
END_FOR
contains := FALSE;
END_METHOD

METHOD get : POINTER TO BYTE
VAR_INPUT
	index : INT;
END_VAR
VAR_OUTPUT
	getSize : LINT;
END_VAR
IF length = 0 OR index < 0 OR index >= length THEN
	get := 0;
	getSize := 0;
ELSE
	elements.GetEntry(diIndex := index, pResultEntry := ADR(get));
	elementSizes.GetEntry(diIndex := index, pResultEntry := ADR(getSize));
END_IF
END_METHOD

METHOD isEmpty : BOOL
VAR_INPUT
END_VAR
isEmpty := length = 0;
END_METHOD

METHOD poll : POINTER TO BYTE
VAR_OUTPUT
	getSize : LINT;
END_VAR
poll := get(index := 0, getSize => getSize);

IF length > 0 THEN
	elements.RemoveEntry(diIndex := 0);
	elementSizes.RemoveEntry(diIndex := 0);
	
	length := length - 1;
END_IF
END_METHOD

METHOD push : BOOL
VAR_INPUT
	value : ANY;
END_VAR
VAR
	temp : POINTER TO BYTE;
END_VAR
temp := __NEW(BYTE, TO_UDINT(value.diSize));
MEMCPY(temp, value.pValue, TO_UDINT(value.diSize));

elements.AddEntryPtr(pEntry := temp);
elementSizes.AddEntry(pEntry := ADR(value.diSize));

length := length + 1;
END_METHOD

METHOD set : BOOL
VAR_INPUT
	i : INT;
	value : ANY;
END_VAR
VAR
	temp : POINTER TO BYTE;
	tempSize : UDINT;
END_VAR
IF length = 0 THEN
	RETURN;
END_IF

IF i >= 0 AND i < length THEN
	temp := get(i);
	__DELETE(temp);
	
	tempSize := TO_UDINT(value.diSize);
	temp := __NEW(BYTE, tempSize);
	MEMCPY(temp, value.pValue, tempSize);

	elements.SetEntryPtr(i, ADR(temp));
	elementSizes.SetEntry(i, ADR(tempSize)); 
	set := TRUE;
END_IF
END_METHOD

METHOD size : INT
size := length;
END_METHOD

END_FUNCTION_BLOCK

// ---- COMMs_TCP/Types/TcpDataQueue.TcPOU
{attribute 'call_after_init'}
FUNCTION_BLOCK TcpDataQueue
VAR
	elements : FB_BA_DynamicArray := (uiEntrySize := SIZEOF(POINTER TO TcpData), uiMinExpCount := GVL.initArraySize); 
	length : INT := 0;
	
	entrySize : UDINT;
END_VAR
(*
this container stores dynamically generated AdsData Structs
AdsData to be added are passed by reference, then this function block allocates a structure to be stored
AdsData are get() by reference and poll() by value
*)

METHOD clear : BOOL
VAR
	i : INT;
	temp : REFERENCE TO TcpData;
	tempAdr : POINTER TO TcpData;
END_VAR
FOR i:=0 TO length-1 BY 1 DO
	temp := get(index := i, getSize => );
	tempAdr := ADR(temp);
	__DELETE(tempAdr);
END_FOR

elements.Reset();
length := 0;
END_METHOD

METHOD contains : BOOL //check contents, not pointer value
VAR_INPUT
	value : REFERENCE TO TcpData;
END_VAR
VAR_OUTPUT
	atIndex : INT;
END_VAR
VAR
	temp : REFERENCE TO TcpData;
	i : INT;
END_VAR
IF length = 0 THEN
	contains := FALSE;
	RETURN;
END_IF

FOR i:=0 TO length-1 BY 1 DO
	temp := get(index := i, getSize => );
	
	IF 
		SIZEOF(value) = entrySize AND //same size
		MEMCMP(ADR(temp), ADR(value), SIZEOF(entrySize)) = 0 //same data
	THEN
		contains := TRUE;
		atIndex := i;
		RETURN;
	END_IF
	
END_FOR
contains := FALSE;
END_METHOD

METHOD get : REFERENCE TO TcpData
VAR_INPUT
	index : INT;
END_VAR
VAR_OUTPUT
	getSize : UDINT;
END_VAR
IF length = 0 OR index < 0 OR index >= length THEN
	getSize := 0;
ELSE
	elements.GetEntry(diIndex := index, pResultEntry := ADR(get));
	getSize := SIZEOF(get);
END_IF
END_METHOD

METHOD isEmpty : BOOL
VAR_INPUT
END_VAR
isEmpty := length = 0;
END_METHOD

METHOD poll : TcpData
VAR_OUTPUT
	getSize : UDINT;
END_VAR
IF length > 0 THEN
	poll := get(index := 0, getSize => getSize);
	elements.RemoveEntry(diIndex := 0);
	
	length := length - 1;
END_IF
END_METHOD

METHOD push : BOOL
VAR_INPUT
	value : REFERENCE TO TcpData;
END_VAR
VAR
	temp : POINTER TO TcpData;
END_VAR
temp := __NEW(TcpData);
temp^ := value;

elements.AddEntryPtr(pEntry := temp);

length := length + 1;
END_METHOD

METHOD set : BOOL
VAR_INPUT
	i : INT;
	value : REFERENCE TO TcpData;
END_VAR
VAR
	temp : REFERENCE TO TcpData;
END_VAR
IF length = 0 THEN
	RETURN;
END_IF

IF i >= 0 AND i < length THEN
	temp REF= get(i);
	temp := value;
	
	set := TRUE;
END_IF
END_METHOD

{attribute 'call_after_init'}
METHOD setup : BOOL
VAR_INPUT
END_VAR
entrySize := SIZEOF(TcpData);
END_METHOD

METHOD size : INT
size := length;
END_METHOD

END_FUNCTION_BLOCK

// ---- DUTs/Containers/PtrQueue.TcPOU
FUNCTION_BLOCK PtrQueue EXTENDS Queue //stores pointers to bundles, not the bundles themselves
VAR_INPUT
	
END_VAR
VAR
	elements : FB_BA_DynamicArray := (uiEntrySize := SIZEOF(PVOID), uiMinExpCount := GVL.initArraySize);
	//length : USINT := 0;
END_VAR

METHOD get : PVOID;
VAR_INPUT
	i : UINT;
END_VAR
elements.GetEntry(diIndex := i, pResultEntry := ADR(get));
END_METHOD

METHOD isEmpty : BOOL
VAR_INPUT
END_VAR
isEmpty := (elements.diCount = 0);
END_METHOD

METHOD poll : PVOID;
VAR_INST
	i : UINT;
END_VAR
poll := get(i := 0);
elements.RemoveEntry(diIndex := 0);
//length := length - 1;
END_METHOD

METHOD push : BOOL
VAR_INPUT
	value : PVOID;
END_VAR
elements.AddEntryPtr(pEntry := value);
//length := length + 1;
push := TRUE;
END_METHOD

METHOD size : DINT
VAR_INPUT
END_VAR
size := elements.diCount;
END_METHOD

END_FUNCTION_BLOCK

// ---- POUs/CallHardware.TcPOU
PROGRAM CallHardware
VAR
	i : DINT;
END_VAR

//conveyors
ForceSetLifterConveyors();

FOR i:=0 TO 20 BY 1 DO
	allConveyors[i]();
END_FOR

//robots
FOR i:=1 TO 6 BY 1 DO
	robots[i]();
END_FOR

//A23
wrapperA23();

//A22
cardboardSkidLeft();
cardboardSkidRight();
cornerGuardMagazineLeft();
cornerGuardMagazineRight();

insertionA22Left();
insertionA22Right();
insertionA22Bottom();
wrapperA22();

//A21
chipboardSkidLeft();
chipboardSkidRight();

woodBunkMagazineLeft();
woodBunkMagazineRight();

stagingTableLeft();
stagingTableRight();

strapperA21();

insertionA21Left();
insertionA21Right();
insertionA21Bottom();

(*
//paper
Hardware.wrapperPaper();

//cardboard + corner guard
FOR i:=Surface.LEFT TO Surface.RIGHT BY 1 DO
	Hardware.insertionCardboardCornerGuardSides[i]();
END_FOR
Hardware.wrapperCardboardCornerguard();

//wood bunk
FOR i:=Surface.LEFT TO Surface.RIGHT BY 1 DO
	Hardware.insertionWoodBunkSides[i]();
	Hardware.stagingTable[i]();
	Hardware.woodBunkMagazine[i]();
END_FOR

Hardware.strapper();
*)

END_PROGRAM

// ---- POUs/Helper Functions/Misc/ForceSetLifterConveyors.TcPOU
FUNCTION ForceSetLifterConveyors : BOOL
VAR
	i : INT;
	temp : REFERENCE TO BOOL;
END_VAR

(*
lifter conveyors:
	5..7
	//add more here
*)

FOR i:=5 TO 7 BY 1 DO
	temp REF= allConveyors[i].hasLifter;
	temp := TRUE;
END_FOR

END_FUNCTION

// ---- POUs/ConveyorControl.TcPOU
PROGRAM ConveyorControl
VAR
	conveyors : POINTER TO Conveyor;
	spoolTimer : TON;
	
	i : INT;
END_VAR
VAR CONSTANT
	spoolSpacing : TIME := T#100MS;
END_VAR

conveyors := ADR(Hardware.allConveyors);

//use one or the other, not both
linkCompute();
//cyclicCompute();

spoolTimer(IN:= , PT:= spoolSpacing, Q=> , ET=> );
spoolTimer.IN := TRUE;
IF
	(conveyors[i].request = ConveyorMode.FORWARD OR conveyors[i].request = ConveyorMode.BACKWARD) AND //conveyor requests motion
	conveyors[i].request <> conveyors[i].operation AND //conveyor request differs from current operation
	spoolTimer.Q //ready to spool
THEN
	//spool up conveyor
	i := i + 1;
	spoolTimer.IN := FALSE;
END_IF

METHOD PRIVATE cyclicCompute : BOOL
VAR
	i : INT;
END_VAR
(*
cyclic computation method
if the last conveyor has the highest priority in a long link, it will take several cycles to reach the other end
*)

FOR i:=Hardware.numConveyors TO 1 BY -1 DO
	IF NOT conveyors[i].occupied() THEN
		//turn conveyor off, but do not change request mode
		conveyors[i].setOperation(ConveyorMode.IDLE);
		CONTINUE;
	END_IF
	
	//conveyor is occupied:
	IF i = Hardware.numConveyors THEN //no next conveyor
		conveyors[i].setOperation( MAX(conveyors[i].request, conveyors[i-1].operation) );
	
	ELSIF i < Hardware.numConveyors AND i > 1 THEN
		
		IF conveyors[i+1].occupied() THEN //next conveyor is occupied
			conveyors[i].setOperation( MAX(conveyors[i+1].operation, conveyors[i].request) );
		END_IF
		
	END_IF
	
END_FOR
END_METHOD

METHOD PRIVATE linkCompute : BOOL
VAR
	i : INT;
	j : INT;
	
	linkStart : INT := -1;
	linkEnd : INT := -1;
	
	priorityInLink : ConveyorMode;
END_VAR
(*
link interation method 
slower, but will correctly set all operations every cycle
*)
FOR i:=1 TO Hardware.numConveyors BY 1 DO
	IF conveyors[i].occupied() THEN
		
		IF linkStart = -1 THEN
			linkStart := i;
		END_IF
		
		priorityInLink := MAX(priorityInLink, conveyors[i].request);
		linkEnd := i;
		
	ELSIF linkStart <> -1 AND linkEnd <> -1 THEN //set all conveyor operations to priorityInLink
		linkEnd := i-1;
		
		FOR j:=linkStart TO linkEnd BY 1 DO
			conveyors[j].setOperation(priorityInLink);
		END_FOR
		
		linkStart := -1;
		linkEnd := -1;
		priorityInLink := ConveyorMode.IDLE;
		
		CONTINUE;
	END_IF
	
END_FOR

linkEnd := linkEnd - 1; //remove residual increment from for loop's failed iteration
IF linkStart > -1 AND linkEnd > -1 THEN
	FOR j:=linkStart TO linkEnd BY 1 DO
		conveyors[j].setOperation(priorityInLink);
	END_FOR
END_IF
END_METHOD

END_PROGRAM

// ---- POUs/Helper Functions/Document/VisionJsonParser.TcPOU
PROGRAM VisionJsonParser
VAR_IN_OUT CONSTANT
	jsonString : STRING(1000);
END_VAR
VAR		
	fbJson : FB_JsonDomParser;
	jsonDoc : SJsonValue;
	
	jsonMaterialID : SJsonValue;
	jsonCheckFor : SJsonValue;
	jsonCameraNumber : SJsonValue;
	jsonSuccessFlag : SJsonValue;
	jsonOrientAdjust : ARRAY[0..2] OF SJsonValue;
	
	i : INT;
END_VAR
VAR_OUTPUT
	visionData : VisionFrame;
END_VAR
VAR CONSTANT
	x : INT := 0;
	y : INT := 1;
	z : INT := 2;
END_VAR

jsonDoc := fbJson.ParseDocument(jsonString);

IF fbJson.HasMember(jsonDoc, 'MaterialID') THEN
	jsonMaterialID := fbJson.FindMember(jsonDoc, 'MaterialID');
END_IF
IF fbJson.HasMember(jsonDoc, 'CheckFor') THEN
	jsonCheckFor := fbJson.FindMember(jsonDoc, 'CheckFor');
END_IF
IF fbJson.HasMember(jsonDoc, 'CameraNumber') THEN
	jsonCameraNumber := fbJson.FindMember(jsonDoc, 'CameraNumber');
END_IF

IF fbJson.HasMember(jsonDoc, 'SuccessFlag') THEN
	jsonSuccessFlag := fbJson.FindMember(jsonDoc, 'SuccessFlag');
END_IF
IF fbJson.HasMember(jsonDoc, 'OrientAdjustX') THEN
	jsonOrientAdjust[x] := fbJson.FindMember(jsonDoc, 'OrientAdjustX');
END_IF
IF fbJson.HasMember(jsonDoc, 'OrientAdjustY') THEN
	jsonOrientAdjust[y] := fbJson.FindMember(jsonDoc, 'OrientAdjustY');
END_IF
IF fbJson.HasMember(jsonDoc, 'OrientAdjustZ') THEN
	jsonOrientAdjust[z] := fbJson.FindMember(jsonDoc, 'OrientAdjustZ');
END_IF

visionData.MaterialID := fbJson.GetString(jsonMaterialID);
visionData.CheckFor := fbJson.GetString(jsonCheckFor);
visionData.CameraNumber := fbJson.GetInt(jsonCameraNumber);

visionData.SuccessFlag := fbJson.GetInt(jsonSuccessFlag);
visionData.OrientAdjustX := fbJson.GetDouble(jsonOrientAdjust[x]);
visionData.OrientAdjustY := fbJson.GetDouble(jsonOrientAdjust[y]);
visionData.OrientAdjustZ := fbJson.GetDouble(jsonOrientAdjust[z]);

END_PROGRAM

// ---- POUs/Helper Functions/Material Functions/GetPositionMasterLength.TcPOU
FUNCTION GetPositionMasterLength : REAL
VAR_INPUT
	currentPair : REFERENCE TO PositionMaterials;
END_VAR
VAR
	topLength : REAL;
	leftLength : REAL;
	rightLength : REAL;
	bottomLength : REAL;
	
	topLeftLength : REAL;
	topRightLength : REAL;
	bottomLeftLength : REAL;
	bottomRightLength : REAL;
END_VAR

topLength := GetMaterialLength(currentPair.top);
leftLength := GetMaterialLength(currentPair.left);
rightLength := GetMaterialLength(currentPair.right);
bottomLength := GetMaterialLength(currentPair.bottom);

topLeftLength := GetMaterialLength(currentPair.topLeft);
topRightLength := GetMaterialLength(currentPair.topRight);
bottomLeftLength := GetMaterialLength(currentPair.bottomLeft);
bottomRightLength := GetMaterialLength(currentPair.bottomRight);

GetPositionMasterLength := MAX(topLength, leftLength, rightLength, bottomLength, topLeftLength, topRightLength, bottomLeftLength, bottomRightLength);

END_FUNCTION

// ---- POUs/Helper Functions/Material Functions/GetMaterialLength.TcPOU
FUNCTION GetMaterialLength : REAL
VAR_INPUT
	material : STRING;
END_VAR
VAR
	i : INT;
END_VAR

FOR i:=0 TO GVL.numMaterials BY 1 DO
	IF GVL.allMaterials[i].code = material THEN
		getMaterialLength := GVL.allMaterials[i].length;
		RETURN;
	END_IF
END_FOR
//otherwise, return 0
GetMaterialLength := 0;

END_FUNCTION

// ---- POUs/Helper Functions/Material Functions/MatchesMaterialType.TcPOU
FUNCTION MatchesMaterialType : BOOL
VAR_INPUT
	pair : REFERENCE TO PositionMaterials;
	materialType : STRING;
END_VAR
VAR
END_VAR

MatchesMaterialType :=
	FIND(pair.top, materialType) > 0 AND
	FIND(pair.left, materialType) > 0 AND
	FIND(pair.right, materialType) > 0 AND
	FIND(pair.bottom, materialType) > 0 AND
	
	FIND(pair.topLeft, materialType) > 0 AND
	FIND(pair.topRight, materialType) > 0 AND
	FIND(pair.bottomLeft, materialType) > 0 AND
	FIND(pair.bottomRight, materialType) > 0 ;

END_FUNCTION

// ---- POUs/Helper Functions/Misc/SizeCheck.TcPOU
PROGRAM SizeCheck
VAR
	bundleSize : ULINT;
	adsDataSize : ULINT;
	tcpDataSize : ULINT;
	
	thousandByteSize : ULINT;
	buffer : ARRAY[0..1000] OF BYTE;
	
	bitArr : ARRAY[1..64] OF ONE_BIT;
	bitArrSize : ULINT;
END_VAR

bundleSize := SIZEOF(Bundle);
adsDataSize := SIZEOF(AdsData);
tcpDataSize := SIZEOF(TcpData);

thousandByteSize := SIZEOF(buffer);

bitArrSize := SIZEOF(bitArr);

END_PROGRAM

// ---- POUs/MAIN.TcPOU
PROGRAM MAIN
VAR_OUTPUT //globally readable, but only modifiable by MAIN
	outputBuffer : ARRAY[Surface.LEFT..Surface.RIGHT] OF Bundle;
	outputBufferPass, outputBufferFail : Bundle;
	numOutputBundles : USINT := 0;
	
	bundleIn : Bundle;
	bundleOut : Bundle;
	
	ready : BOOL;
	busy : BOOL;
	done : BOOL;
	error : BOOL;
	backlog : BOOL;
	
	localTime : TIMESTRUCT;
	pause : BOOL;
END_VAR
VAR
	removeBundle AT %I* : ARRAY[Surface.LEFT..Surface.RIGHT] OF BOOL;
	clearPassBuffer, clearFailBuffer AT %I* : BOOL;
	receiverStruct : AdsData;
	
	//ETA is not strictly required, area will process bundle even if it is not in ETA arrays
	expectedBundles : ARRAY[0..GVL.maxQueue] OF STRING; //bundles expected to arrive
	expectedArrivals : ARRAY[0..GVL.maxQueue] OF TIMESTRUCT; //bundles expected to arrive
	numEtaBundles : INT;
	
	//parallel arrays - bundle, bypass
	numBundlesQueue : INT;
	bundlesQueue : ARRAY[0..GVL.maxQueue] OF Bundle;
	bundlesBypass : ARRAY[0..GVL.maxQueue] OF BOOL;
	
	//spacerRecollector : PackagerFreeAsync;
	paperSection : PaperEx;
	cardboardCornerGuardSection : CardboardCornerGuardEx;
	chipboardSection : ChipboardEx;
	woodBunkSection : WoodBunkEx;
	outputSection : AreaOutputEx;
	run : ARRAY[0..SectionEnum.size] OF BOOL := [6(TRUE)];
	
	fbLocalSystemTime : FB_LocalSystemTime;
	fbEventLogger : SqlDatabaseAccessor;
	
	start : BOOL;
	
	processingMode : (PARALLEL, SINGLE, SERIAL, CLEAR);
	requestedMode : (PARALLEL, SINGLE, SERIAL, CLEAR);
	serialSection : REFERENCE TO SectionEx;
END_VAR
VAR //these variables are only tracked for HMI
	sectionsBusy : ARRAY[0..SectionEnum.size] OF BOOL;
	sectionsIterator : ARRAY[0..SectionEnum.size] OF INT;
END_VAR
VAR CONSTANT
	numSections : INT := 6;
	maxOutputBundles : USINT := 3;
END_VAR

demoHMI();

SizeCheck();
getLocalTime();

AdsClient( //PLC-PLC comms
	ServerNetId:= , 
	ServerPort:= , 
	bBusy=> , 
	err=> , 
	errid=> , 
	localPrgName=> , 
	localNetId=> , 
	localPort=> , 
	socketReady=> , 
	remoteAccessPrefix=> );
	
TcpServer1Vision( //PLC-Vision comms
	ServerNetId:= , 
	ServerAdr:= , 
	ServerPort:= , 
	busy=> , 
	error=> , 
	errorId=> , 
	bytesReceived=> , 
	connected=> , 
	receiveStruct=> );
	
IF NOT ( enableHardware() AND initialize() ) OR pause THEN
	RETURN;	
END_IF

//THIS MUST BE CALLED FIRST
CallHardware();
ConveyorControl();

IF AdsClient.fetchData(receiverStruct) THEN
	interpretTransmission(receiverStruct);
END_IF


IF ready AND BundleIsValid(bundleIn) THEN
	receive();
END_IF


IF NOT busy THEN
	processingMode := requestedMode;
END_IF
requestMode();

IF clearPassBuffer OR clearFailBuffer THEN
	transfer();
	shiftBundles();
END_IF

ready := paperSection.ready; //if A2 is not ready, dispatch controller must block operator from sending bundles here
busy := paperSection.busy OR cardboardCornerGuardSection.busy OR chipboardSection.busy OR woodBunkSection.busy OR outputSection.busy;
done := outputSection.done;
backlog := numBundlesQueue > 5;



fbEventLogger();

METHOD demoHMI : BOOL
VAR
	i : INT;
END_VAR
IF NOT start THEN //for HMI testing only, remove for production
	FOR i:=0 TO GVL.maxQueue BY 1 DO
		bundlesQueue[i].id := TO_STRING(i);
	END_FOR
	
	start := TRUE;
END_IF
END_METHOD

METHOD PRIVATE enableHardware : BOOL
VAR
	iCardboardSlot : CornerGuard := 1;
	iCornerGuardSlot : Cardboard := 1;
	iChipboardSlot : Chipboard := 1;
	iWoodBunkSlot : WoodBunk := 1;
	
	slotsArr : ARRAY[1..GVL.maxQueue] OF STRING;
	
	i : INT;
END_VAR
FOR iCardboardSlot:=1 TO Cardboard.size-1 BY 1 DO
	slotsArr[iCardboardSlot] := TO_STRING(iCardboardSlot);
END_FOR
cardboardSkidLeft.setupSlots(slotsArr);
cardboardSkidRight.setupSlots(slotsArr);


FOR iCornerGuardSlot:=1 TO CornerGuard.size-1 BY 1 DO
	slotsArr[iCornerGuardSlot] := TO_STRING(iCornerGuardSlot);
END_FOR
cornerGuardMagazineLeft.setupSlots(slotsArr);
cornerGuardMagazineRight.setupSlots(slotsArr);


FOR iChipboardSlot:=1 TO Chipboard.size-1 BY 1 DO
	slotsArr[iChipboardSlot] := TO_STRING(iChipboardSlot);
END_FOR
chipboardSkidLeft.setupSlots(slotsArr);
chipboardSkidRight.setupSlots(slotsArr);


FOR iWoodBunkSlot:=1 TO WoodBunk.size-1 BY 1 DO
	slotsArr[iWoodBunkSlot] := TO_STRING(iWoodBunkSlot);
END_FOR
woodBunkMagazineLeft.setupSlots(slotsArr);
woodBunkMagazineRight.setupSlots(slotsArr);


insertionA22Left.enable := TRUE;
insertionA21Left.enable := TRUE;

enableHardware := TRUE;
END_METHOD

METHOD PRIVATE getLocalTime : BOOL
fbLocalSystemTime(
	sNetID:= '', 
	bEnable:= TRUE, 
	dwCycle:= , 
	dwOpt:= , 
	tTimeout:= , 
	bValid=> , 
	systemTime=> localTime, 
	tzID=> );
	
getLocalTime := TRUE;
END_METHOD

METHOD PRIVATE initialize : BOOL
VAR
	i : INT;
	temp : POINTER TO BOOL;
END_VAR
paperSection.connectTo(ADR(cardboardCornerGuardSection));
cardboardCornerGuardSection.connectTo(ADR(chipboardSection));
chipboardSection.connectTo(ADR(woodBunkSection));
woodBunkSection.connectTo(ADR(outputSection));

paperSection.sectionID := SectionEnum.PAPER;
cardboardCornerGuardSection.sectionID := SectionEnum.CARDBOARD_CORNERGUARD;
chipboardSection.sectionID := SectionEnum.CHIPBOARD;
woodBunkSection.sectionID := SectionEnum.WOOD_BUNK;
outputSection.sectionID := SectionEnum.OUTPUT;

(*
	paperSection.accessNextSection := ADR(cardboardCornerGuardSection);
	cardboardCornerGuardSection.accessNextSection := ADR(chipboardSection);
	chipboardSection.accessNextSection := ADR(woodBunkSection);
	woodBunkSection.accessNextSection := ADR(outputSection);
	outputSection.accessNextSection := 0;
	
	outputSection.accessPrevSection := woodBunkSection;
	woodBunkSection.accessPrevSection := chipboardSection;
	chipboardSection.accessPrevSection := cardboardCornerGuardSection;
	cardboardCornerGuardSection.accessPrevSection := paperSection;
	paperSection.accessPrevSection := 0;
*)

(*
	12, 20	entry + paper
	9, 11	cardboard + corner guard
	5, 8	chipboard + wood bunk
	1, 4 	output buffer
	
	0, 0 	spacer recollector (possibly obsolete)
*)
ForceSetLifterConveyors();

paperSection.assignConveyors(12, 20);
cardboardCornerGuardSection.assignConveyors(9, 11);
chipboardSection.assignConveyors(5, 8);
woodBunkSection.assignConveyors(5, 8);
outputSection.assignConveyors(1, 4);

initialize := TRUE;
END_METHOD

METHOD PRIVATE interpretTransmission : BOOL
VAR_INPUT
	data : REFERENCE TO AdsData;
END_VAR
VAR
	i : INT;
END_VAR
CASE data.description OF
	EventsEnum.BUNDLE_IN:
		MEMCPY(ADR(bundleIn), ADR(data.binaryData), SIZEOF(bundleIn));
			
	EventsEnum.BUNDLE_ETA:
		MEMCPY(ADR(expectedBundles[numEtaBundles]), ADR(data.binaryData), SIZEOF(expectedBundles[numEtaBundles]));
		expectedArrivals[numEtaBundles] := data.timestamp;
		
END_CASE
END_METHOD

METHOD PRIVATE process : BOOL
(*
full parallel processsing
all sections may operate concurrently on any bundle
*)
paperSection(
	enable:= run[SectionEnum.PAPER], 
	bundlesQueue:= bundlesQueue, 
	bundlesBypass:= bundlesBypass,
	bundleOut=> , 
	bypass=> , 
	ready=> , 
	busy=> sectionsBusy[SectionEnum.PAPER], 
	done=> , 
	error=> , 
	backlog=> ,
	iBundle=> sectionsIterator[SectionEnum.PAPER],
	iPair=> );
	
cardboardCornerGuardSection(
	enable:= run[SectionEnum.CARDBOARD_CORNERGUARD],
	bundlesQueue:= bundlesQueue, 
	bundlesBypass:= bundlesBypass,
	bundleOut=> ,
	bypass=> , 
	ready=> , 
	busy=> sectionsBusy[SectionEnum.CARDBOARD_CORNERGUARD], 
	done=> , 
	error=> , 
	backlog=> ,
	iBundle=> sectionsIterator[SectionEnum.CARDBOARD_CORNERGUARD],
	iPair=> );

chipboardSection(
	enable:= run[SectionEnum.CHIPBOARD],
	bundlesQueue:= bundlesQueue, 
	bundlesBypass:= bundlesBypass, 
	bundleOut=> ,
	bypass=> , 
	ready=> , 
	busy=> sectionsBusy[SectionEnum.CHIPBOARD], 
	done=> , 
	error=> , 
	backlog=> ,
	iBundle=> sectionsIterator[SectionEnum.CHIPBOARD],
	iPair=> );

woodBunkSection(
	enable:= run[SectionEnum.WOOD_BUNK],
	bundlesQueue:= bundlesQueue, 
	bundlesBypass:= bundlesBypass, 
	bundleOut=> ,
	bypass=> , 
	ready=> , 
	busy=> sectionsBusy[SectionEnum.WOOD_BUNK], 
	done=> , 
	error=> , 
	backlog=> ,
	iBundle=> sectionsIterator[SectionEnum.WOOD_BUNK],
	iPair=> );
	
outputSection(
	enable:= run[SectionEnum.OUTPUT],
	bundlesQueue:= bundlesQueue, 
	bundlesBypass:= bundlesBypass,
	outputBuffer:= outputBuffer,
	bundleOut=> , 
	bypass=> , 
	ready=> , 
	busy=> sectionsBusy[SectionEnum.OUTPUT],
	done=> , 
	error=> , 
	backlog=> ,
	iBundle=> sectionsIterator[SectionEnum.OUTPUT],
	iPair=> );
END_METHOD

{attribute 'TcRpcEnable'}
METHOD PRIVATE receive : BOOL
VAR
	i : INT;
	shiftIndex : INT := -1;
	invalidBundle : Bundle;
END_VAR
FOR i:=0 TO GVL.maxQueue BY 1 DO //find the bundle in the ETA queue
	IF expectedBundles[i] = bundleIn.id THEN
		shiftIndex := i;
		EXIT;
	END_IF
END_FOR

IF shiftIndex > -1 THEN //if the bundle is found in the ETA queue, shift everything down
	MEMMOVE(
		ADR(expectedBundles[shiftIndex]), 
		ADR(expectedBundles[shiftIndex + 1]), 
		SIZEOF(STRING) * TO_UINT(GVL.maxQueue - shiftIndex));
		
	MEMMOVE(
		ADR(expectedArrivals[shiftIndex]), 
		ADR(expectedArrivals[shiftIndex + 1]), 
		SIZEOF(TIMESTRUCT) * TO_UINT(GVL.maxQueue - shiftIndex) );
		
	numEtaBundles := numEtaBundles - 1;
END_IF

FOR i:=0 TO GVL.maxQueue BY 1 DO
	IF BundleIsValid(bundlesQueue[i]) AND NOT bundlesBypass[i] THEN
		bundlesQueue[i] := bundleIn;
		bundlesBypass[i] := FALSE;
		
		receive := TRUE;
		RETURN;
	END_IF
END_FOR

IF NOT receive THEN
	error := TRUE;
END_IF
END_METHOD

METHOD requestMode : BOOL
CASE requestedMode OF
	PARALLEL:
		//backlog := numBundlesQueue >= 5;
		
	SINGLE:
		backlog := numBundlesQueue >= 1;
		
	SERIAL:
		backlog := numBundlesQueue >= 1;
		
	CLEAR:
		backlog := numBundlesQueue > 0;
		
END_CASE

CASE processingMode OF //run stations
	PARALLEL:
		process();
		backlog := numBundlesQueue >= 5;
		
	SINGLE:
		singleProcess();
		backlog := numBundlesQueue >= 1;
		
	SERIAL:
		serialProcess();
		backlog := numBundlesQueue >= 1;
		
	CLEAR:
		backlog := numBundlesQueue > 0;
		//stop processing
		
END_CASE
END_METHOD

METHOD serialProcess : BOOL
VAR_INPUT
END_VAR
(*
sections process bundles 1 by 1 in order
only 1 bundle allowed in the section at a time
*)
IF NOT __ISVALIDREF(serialSection) THEN
	serialSection REF= PaperSection;
END_IF

serialSection(
	enable:= TRUE, 
	sectionID:= , 
	bundlesQueue:= bundlesQueue, 
	bundlesBypass:= bundlesBypass, 
	bundleOut=> , 
	bypass=> , 
	ready=> , 
	busy=> , 
	done=> , 
	error=> , 
	backlog=> , 
	iBundle=> , 
	iPair=> );
	
IF serialSection.done THEN
	serialSection REF= serialSection.accessNextSection^;
END_IF
END_METHOD

METHOD shiftBundles : BOOL
VAR_INPUT
END_VAR
//shift down parallel arrays
MEMMOVE(ADR(bundlesQueue[0]), ADR(bundlesQueue[1]), SIZEOF(Bundle) * TO_UINT(GVL.maxQueue));
MEMMOVE(ADR(bundlesBypass[0]), ADR(bundlesBypass[1]), SIZEOF(BOOL) * TO_UINT(GVL.maxQueue));

//decrement each section's iterator to realign with their correct bundle
paperSection.shiftIterator();
cardboardCornerGuardSection.shiftIterator();
chipboardSection.shiftIterator();
woodBunkSection.shiftIterator();
outputSection.shiftIterator();
END_METHOD

METHOD singleProcess : BOOL
VAR_INPUT
END_VAR
(*
all sections may operate on a bundle as they arrive
only 1 bundle may enter the area at a time
*)
END_METHOD

METHOD PRIVATE transfer : BOOL
VAR
	i : INT;
END_VAR
//send TCP/ADS transmission back to Dispatch once bundle is removed from the plant

IF clearPassBuffer THEN
	fbEventLogger.queueEvent(event:= EventsEnum.BUNDLE_OUT); //modify to include bundle ID
	outputBufferPass := GVL.nullBundle;
END_IF

IF clearFailBuffer THEN
	fbEventLogger.queueEvent(event:= EventsEnum.BUNDLE_OUT); //modify to include bundle ID
	outputBufferFail := GVL.nullBundle;
END_IF
END_METHOD

END_PROGRAM

// ---- Sections/Concrete/PaperEx.TcPOU
FUNCTION_BLOCK PaperEx EXTENDS SectionEx
VAR
	robotLeft, robotRight : REFERENCE TO Robot;
	wrapper : REFERENCE TO WrapMachine;
END_VAR
VAR
	paperConveyorPos : REAL;
	
	robotLeftOutputs, robotRightOutputs : ARRAY[1..50] OF INT;
	
	iTop : USINT;
	iLeft : USINT;
	iRight : USINT;
	iBottom : USINT;
	
	tempConveyorModes : ARRAY[0..4] OF INT; //conveyor enum
	tempConveyorModeTop : INT;
	tempConveyorModeLeft : INT;
	tempConveyorModeRight : INT;
	tempConveyorModeBottom : INT;
END_VAR

entryRefPos := paperConveyorPos;
exitRefPos := paperConveyorPos;

SUPER^();

METHOD changeRobotsEOAT : BOOL
VAR_INPUT
END_VAR
IF robotLeft.tool <> sectionID THEN
	MEMSET(ADR(robotLeftOutputs), 0, SIZEOF(robotLeftOutputs));
	robotLeftOutputs[1] := A21.TOOL_CHANGE_CHIPBOARD;
	robotLeft.setParamsAndWait(robotLeftOutputs);
END_IF

IF robotRight.tool <> sectionID THEN
	MEMSET(ADR(robotRightOutputs), 0, SIZEOF(robotRightOutputs));
	robotRightOutputs[1] := A21.TOOL_CHANGE_CHIPBOARD;
	robotRight.setParamsAndWait(robotRightOutputs);
END_IF

changeRobotsEOAT := robotLeft.tool = sectionID AND robotRight.tool = sectionID;
END_METHOD

METHOD cutPaper : BOOL
VAR_IN_OUT
	tempPaperConveyorOps : ARRAY[*] OF INT; //conveyor enum
END_VAR
VAR_INPUT
	iTop : REFERENCE TO USINT;
	iLeft : REFERENCE TO USINT;
	iRight : REFERENCE TO USINT;
	iBottom : REFERENCE TO USINT;
END_VAR
VAR_INST
	cmdSent : ARRAY[0..4] OF BOOL;
	i : INT;
END_VAR
IF iTop < GVL.maxPairs THEN
	IF paperConveyorPos >= currentBundle.paperTop[iTop].endPos THEN
		IF NOT cmdSent[Surface.TOP] THEN
			tempPaperConveyorOps[Surface.TOP] := ConveyorMode.STOP;
			//instruction - cut paper
			
			IF TRUE(*instruction completed*) THEN
				cmdSent[Surface.TOP] := TRUE;
				iTop := iTop + 1;
				tempPaperConveyorOps[Surface.TOP] := ConveyorMode.FORWARD;
			END_IF
		END_IF
		
		//otherwise do nothing, paper is already being pulled
	END_IF
END_IF

IF iLeft < GVL.maxPairs THEN
	IF paperConveyorPos = currentBundle.paperLeft[iLeft].endPos THEN
		IF NOT cmdSent[Surface.LEFT] THEN
			tempPaperConveyorOps[Surface.LEFT] := ConveyorMode.STOP;
			//instruction - cut paper
			
			IF TRUE(*instruction completed*) THEN
				cmdSent[Surface.LEFT] := TRUE;
				iLeft := iLeft + 1;
				tempPaperConveyorOps[Surface.LEFT] := ConveyorMode.FORWARD;
			END_IF
		END_IF
		
		//otherwise do nothing, paper is already being pulled
	END_IF
END_IF

IF iRight < GVL.maxPairs THEN
	IF paperConveyorPos = currentBundle.paperRight[iRight].endPos THEN
		IF NOT cmdSent[Surface.RIGHT] THEN
			tempPaperConveyorOps[Surface.RIGHT] := ConveyorMode.STOP;
			//instruction - cut paper
			
			IF TRUE(*instruction completed*) THEN
				cmdSent[Surface.RIGHT] := TRUE;
				iRight := iRight + 1;
				tempPaperConveyorOps[Surface.RIGHT] := ConveyorMode.FORWARD;
			END_IF
		END_IF
		
		//otherwise do nothing, paper is already being pulled
	END_IF
END_IF

IF iBottom < GVL.maxPairs THEN
	IF paperConveyorPos = currentBundle.paperBottom[iBottom].endPos THEN
		IF NOT cmdSent[Surface.BOTTOM] THEN
			tempPaperConveyorOps[Surface.BOTTOM] := ConveyorMode.STOP;
			//instruction - cut paper
			
			IF TRUE(*instruction completed*) THEN
				cmdSent[Surface.BOTTOM] := TRUE;
				iBottom := iBottom + 1;
				tempPaperConveyorOps[Surface.BOTTOM] := ConveyorMode.FORWARD;
			END_IF
		END_IF
		
		//otherwise do nothing, paper is already being pulled
	END_IF
END_IF
END_METHOD

METHOD initHardware : BOOL
conveyors := ADR(allConveyors);
END_METHOD

METHOD PROTECTED load : BOOL
VAR_INPUT
	pair : REFERENCE TO PositionMaterials;
END_VAR
END_METHOD

METHOD placePaperBottom : BOOL
VAR_INPUT
	i : REFERENCE TO USINT; //current interval in the paper recipe array
	tempConveyorMode : INT;
END_VAR
VAR
	currentInterval : REFERENCE TO Interval;
END_VAR
VAR_INST
	step : INT;
END_VAR
IF i >= GVL.maxPairs THEN //already finished iterating
	tempConveyorMode := ConveyorMode.IDLE;
	RETURN;
END_IF

currentInterval REF= currentBundle.paperBottom[i];

CASE step OF
	0: //check validity
		IF currentInterval.startPos = GVL.nullPos THEN
			i := i + 1;
			RETURN;
		END_IF
		
		IF InRange(paperConveyorPos - 0.1, paperConveyorPos + 0.1, currentInterval.startPos, EXCLUSIVE) THEN
			step := 10;
		ELSIF paperConveyorPos > currentInterval.startPos THEN
			tempConveyorMode := ConveyorMode.BACKWARD;
		ELSIF paperConveyorPos < currentInterval.startPos THEN
			tempConveyorMode := ConveyorMode.FORWARD;
		END_IF
				
	10: //pull paper
		IF i < GVL.maxPairs AND paperConveyorPos >= currentInterval.startPos THEN
			tempConveyorMode := ConveyorMode.STOP;
			//instruction - pull roll
			IF TRUE (*instruction finished*) THEN
				step := 20;
				tempConveyorMode := ConveyorMode.FORWARD;
			END_IF
		END_IF
			
	20: //cut paper
		
		
		IF paperConveyorPos >= currentInterval.endPos THEN
			//instruction - cut roll
			IF TRUE (*instruction finished*) THEN
				step := 30;
			END_IF
		END_IF
		
	30: //reset
		tempConveyorMode := ConveyorMode.IDLE;
		i := i + 1;
		step := 0;
END_CASE
END_METHOD

METHOD placePaperLeft : BOOL
VAR_IN_OUT
	i : USINT; //current interval in the paper recipe array
	tempConveyorMode : INT;
END_VAR
VAR
	currentInterval : REFERENCE TO Interval;
END_VAR
VAR_INST
	step : INT;
END_VAR
IF i >= GVL.maxPairs THEN //already finished iterating
	tempConveyorMode := ConveyorMode.IDLE;
	RETURN;
END_IF

currentInterval REF= currentBundle.paperLeft[i];

CASE step OF
	0: //check validity
		IF currentInterval.startPos = GVL.nullPos THEN
			i := i + 1;
			RETURN;
		END_IF
		
		IF InRange(paperConveyorPos - 0.1, paperConveyorPos + 0.1, currentInterval.startPos, EXCLUSIVE) THEN
			step := 10;
		ELSIF paperConveyorPos > currentInterval.startPos THEN
			tempConveyorMode := ConveyorMode.BACKWARD;
		ELSIF paperConveyorPos < currentInterval.startPos THEN
			tempConveyorMode := ConveyorMode.FORWARD;
		END_IF
				
	10: //pull paper
		IF i < GVL.maxPairs AND paperConveyorPos >= currentInterval.startPos THEN
			tempConveyorMode := ConveyorMode.STOP;
			//instruction - pull roll
			IF TRUE (*instruction finished*) THEN
				step := 20;
				tempConveyorMode := ConveyorMode.FORWARD;
			END_IF
		END_IF
			
	20: //cut paper
		
		
		IF paperConveyorPos >= currentInterval.endPos THEN
			//instruction - cut roll
			IF TRUE (*instruction finished*) THEN
				step := 30;
			END_IF
		END_IF
		
	30: //reset
		tempConveyorMode := ConveyorMode.IDLE;
		i := i + 1;
		step := 0;
END_CASE
END_METHOD

METHOD placePaperRight : BOOL
VAR_INPUT
	i : REFERENCE TO USINT; //current interval in the paper recipe array
	tempConveyorMode : INT;
END_VAR
VAR
	currentInterval : REFERENCE TO Interval;
END_VAR
VAR_INST
	step : INT;
END_VAR
IF i >= GVL.maxPairs THEN //already finished iterating
	tempConveyorMode := ConveyorMode.IDLE;
	RETURN;
END_IF

currentInterval REF= currentBundle.paperRight[i];

CASE step OF
	0: //check validity
		IF currentInterval.startPos = GVL.nullPos THEN
			i := i + 1;
			RETURN;
		END_IF
		
		IF InRange(paperConveyorPos - 0.1, paperConveyorPos + 0.1, currentInterval.startPos, EXCLUSIVE) THEN
			step := 10;
		ELSIF paperConveyorPos > currentInterval.startPos THEN
			tempConveyorMode := ConveyorMode.BACKWARD;
		ELSIF paperConveyorPos < currentInterval.startPos THEN
			tempConveyorMode := ConveyorMode.FORWARD;
		END_IF
				
	10: //pull paper
		IF i < GVL.maxPairs AND paperConveyorPos >= currentInterval.startPos THEN
			tempConveyorMode := ConveyorMode.STOP;
			//instruction - pull roll
			IF TRUE (*instruction finished*) THEN
				step := 20;
				tempConveyorMode := ConveyorMode.FORWARD;
			END_IF
		END_IF
			
	20: //cut paper
		
		
		IF paperConveyorPos >= currentInterval.endPos THEN
			//instruction - cut roll
			IF TRUE (*instruction finished*) THEN
				step := 30;
			END_IF
		END_IF
		
	30: //reset
		tempConveyorMode := ConveyorMode.IDLE;
		i := i + 1;
		step := 0;
END_CASE
END_METHOD

METHOD placePaperTop : BOOL
VAR_INPUT
	i : REFERENCE TO USINT; //current interval in the paper recipe array
	tempConveyorMode : INT;
END_VAR
VAR
	currentPair : REFERENCE TO Interval;
END_VAR
VAR_INST
	step : INT;
END_VAR
IF i >= GVL.maxPairs THEN //already finished iterating
	tempConveyorMode := ConveyorMode.IDLE;
	RETURN;
END_IF

currentPair REF= currentBundle.paperTop[i];

CASE step OF
	0: //check validity
		IF currentPair.startPos = GVL.nullPos THEN
			i := i + 1;
			RETURN;
		END_IF
		
		IF directionCheckAndSet(paperConveyorPos, currentPair.startPos) THEN
			step := 10;
		END_IF
				
	10: //pull paper
		IF i < GVL.maxPairs AND paperConveyorPos >= currentPair.startPos THEN
			tempConveyorMode := ConveyorMode.STOP;
			//instruction - pull roll
			IF TRUE (*instruction finished*) THEN
				step := 20;
				tempConveyorMode := ConveyorMode.FORWARD;
			END_IF
		END_IF
			
	20: //cut paper
		
		
		IF paperConveyorPos >= currentPair.endPos THEN
			//instruction - cut roll
			IF TRUE (*instruction finished*) THEN
				step := 30;
			END_IF
		END_IF
		
	30: //reset
		tempConveyorMode := ConveyorMode.IDLE;
		i := i + 1;
		step := 0;
END_CASE
END_METHOD

METHOD PROTECTED process : BOOL
(*
rollPaper(tempConveyorModes, iTop, iLeft, iRight, iBottom);
cutPaper(tempConveyorModes, iTop, iLeft, iRight, iBottom);
*)
placePaperTop(iTop, tempConveyorModeTop);
placePaperLeft(iLeft, tempConveyorModeLeft);
placePaperRight(iRight, tempConveyorModeRight);
placePaperBottom(iBottom, tempConveyorModeBottom);
(*
FOR i:=0 TO 4 BY 1 DO
	requestConveyorMode(MAX(conveyorMode, tempConveyorModes[i]));
END_FOR
*)
setConveyorMode(MAX(tempConveyorModeTop, tempConveyorModeLeft, tempConveyorModeRight, tempConveyorModeBottom));

IF 
	iTop >= GVL.maxPairs AND 
	iLeft >= GVL.maxPairs AND 
	iRight >= GVL.maxPairs AND 
	iBottom >= GVL.maxPairs 
THEN
	setConveyorMode(ConveyorMode.IDLE);
END_IF
END_METHOD

METHOD process2 : BOOL
VAR_INPUT
	//iPair : REFERENCE TO USINT; //redundant, for inheritance compatibility only
END_VAR
VAR
	iTop : REFERENCE TO USINT;
	iLeft : REFERENCE TO USINT;
	iRight : REFERENCE TO USINT;
	iBottom : REFERENCE TO USINT;
	
	tempConveyorModes : ARRAY[0..4] OF INT; //conveyor enum
	
	i : INT;
END_VAR
rollPaper(tempConveyorModes, iTop, iLeft, iRight, iBottom);
cutPaper(tempConveyorModes, iTop, iLeft, iRight, iBottom);

FOR i:=0 TO 4 BY 1 DO
	setConveyorMode(MAX(requestedConveyorMode, tempConveyorModes[i]));
END_FOR

IF 
	iTop >= GVL.maxPairs AND 
	iLeft >= GVL.maxPairs AND 
	iRight >= GVL.maxPairs AND 
	iBottom >= GVL.maxPairs 
THEN
	setConveyorMode(ConveyorMode.IDLE);
END_IF
END_METHOD

METHOD rollPaper : BOOL
VAR_IN_OUT
	tempPaperConveyorOps : ARRAY[*] OF INT; //conveyor enum
END_VAR
VAR_INPUT
	iTop : REFERENCE TO USINT;
	iLeft : REFERENCE TO USINT;
	iRight : REFERENCE TO USINT;
	iBottom : REFERENCE TO USINT;
END_VAR
VAR_INST
	cmdSent : ARRAY[0..4] OF BOOL;
	i : INT;
END_VAR
IF iTop < GVL.maxPairs THEN
	IF paperConveyorPos >= currentBundle.paperTop[iTop].startPos THEN
		IF NOT cmdSent[Surface.TOP] THEN
			tempPaperConveyorOps[Surface.TOP] := ConveyorMode.STOP;
			//instruction - pull paper
			
			IF TRUE(*instruction completed*) THEN
				cmdSent[Surface.TOP] := TRUE;
				tempPaperConveyorOps[Surface.TOP] := ConveyorMode.FORWARD;
			END_IF
		END_IF
		
		//otherwise do nothing, paper is already being pulled
	END_IF
END_IF

IF iLeft < GVL.maxPairs THEN
	IF paperConveyorPos = currentBundle.paperLeft[iLeft].startPos THEN
		IF NOT cmdSent[Surface.LEFT] THEN
			tempPaperConveyorOps[Surface.LEFT] := ConveyorMode.STOP;
			//instruction - pull paper
			
			IF TRUE(*instruction completed*) THEN
				cmdSent[Surface.LEFT] := TRUE;
				tempPaperConveyorOps[Surface.LEFT] := ConveyorMode.FORWARD;
			END_IF
		END_IF
		
		//otherwise do nothing, paper is already being pulled
	END_IF
END_IF

IF iRight < GVL.maxPairs THEN
	IF paperConveyorPos = currentBundle.paperRight[iRight].startPos THEN
		IF NOT cmdSent[Surface.RIGHT] THEN
			tempPaperConveyorOps[Surface.RIGHT] := ConveyorMode.STOP;
			//instruction - pull paper
			
			IF TRUE(*instruction completed*) THEN
				cmdSent[Surface.RIGHT] := TRUE;
				tempPaperConveyorOps[Surface.RIGHT] := ConveyorMode.FORWARD;
			END_IF
		END_IF
		
		//otherwise do nothing, paper is already being pulled
	END_IF
END_IF

IF iBottom < GVL.maxPairs THEN
	IF paperConveyorPos = currentBundle.paperBottom[iBottom].startPos THEN
		IF NOT cmdSent[Surface.BOTTOM] THEN
			tempPaperConveyorOps[Surface.BOTTOM] := ConveyorMode.STOP;
			//instruction - pull paper
			
			IF TRUE(*instruction completed*) THEN
				cmdSent[Surface.BOTTOM] := TRUE;
				tempPaperConveyorOps[Surface.BOTTOM] := ConveyorMode.FORWARD;
			END_IF
		END_IF
		
		//otherwise do nothing, paper is already being pulled
	END_IF
END_IF
END_METHOD

METHOD PROTECTED usesProcess : BOOL
END_METHOD

END_FUNCTION_BLOCK

// ---- Sections/SectionEx.TcPOU
FUNCTION_BLOCK ABSTRACT SectionEx
VAR_INPUT CONSTANT
	enable : BOOL;
	sectionID : SectionEnum;
END_VAR
VAR_IN_OUT
	bundlesQueue : ARRAY[*] OF Bundle;
	bundlesBypass : ARRAY[*] OF BOOL;
END_VAR
VAR_OUTPUT
	bundleOut : Bundle;
	bypass : BOOL;
	
	ready : BOOL;
	busy : BOOL;
	done : BOOL;
	error : BOOL;
	backlog : BOOL;
	
	iBundle : INT(0..GVL.maxQueue);
	iPair : INT(0..GVL.maxPairs);
END_VAR
VAR
	conveyors : POINTER TO Conveyor; //array of conveyors taken from Hardware GVL
	firstConveyor : INT;
	lastConveyor : INT;
END_VAR
VAR	
	currentBundle : REFERENCE TO Bundle;
	currentBypass : REFERENCE TO BOOL;
	
	loaded : BOOL;
	
	entryRefPos : (*REFERENCE TO*) REAL;
	exitRefPos : (*REFERENCE TO*) REAL;
	
	requestedConveyorMode : ConveyorMode;
	
	nextSection : POINTER TO SectionEx;
	prevSection : POINTER TO SectionEx;
	
	occupied : BOOL; //may need to move this to Hardware GVL since this is a sensor
	
	status : SectionStatus; //section status
	
	loadSet : INT;
	loadStepLeft, loadStepRight : INT;
END_VAR
VAR
	
END_VAR
VAR_STAT CONSTANT
	INCLUSIVE : INT := 0;
	EXCLUSIVE : INT := 1;
	COMPLETE : INT := 1030;
END_VAR

(*
currentBundle is the bundle that the section's target bundle and is set if there is a bundle to target
bundleOut is only set once the bundle head starts poking out (status >= ACTIVE)
*)

initHardware();

currentBundle REF= bundlesQueue[iBundle];
currentBypass REF= bundlesBypass[iBundle];
bypass := currentBypass;
	
backlog := iBundle >= GVL.maxQueue;

IF currentBypass THEN
	IF NOT discharge() THEN
		RETURN;
	END_IF
	status := SectionStatus.CLEARING;
END_IF


//set the 3-status register every state
CASE status OF
	SectionStatus.IDLE:
		ready := TRUE;
		busy := FALSE;
		done := done;
		
		IF BundleIsValid(currentBundle) THEN			
			status := SectionStatus.ALIGNING;
		END_IF
	
	SectionStatus.ALIGNING:
		ready := FALSE;
		busy := FALSE;
		done := done;
		
		setConveyorMode(ConveyorMode.FORWARD);
		IF 
			occupied AND
			nextSection <> 0 AND_THEN
			nextSection^.getConveyorMode() = ConveyorMode.BACKWARD
		THEN //section occupied by next section backing up into this section
			status := -100;
			
		ELSIF occupied THEN //section occupied by correct bundle
			//zero the conveyors
			status := SectionStatus.ACTIVE;
			
		END_IF
		
	SectionStatus.ACTIVE:
		ready := FALSE;
		busy := TRUE;
		done := FALSE;
		
		bundleOut := currentBundle;
		
		IF NOT enable THEN
			iPair := 0;
			status := SectionStatus.CLEARING;
			
		//usesProcess may need to be put into I_MaterialSection, TBD
		ELSIF NOT usesProcess() THEN //bundle does not use this section's processes
			iPair := 0;
			status := SectionStatus.CLEARING;
		
		ELSIF currentBypass (*AND_THEN discharge()*) THEN //bundle failed in previous section, discharge this section's materials
			IF discharge() THEN
				iPair := 0;
				status := SectionStatus.CLEARING;
			END_IF
			
		ELSIF process() THEN //bundle recipe completed normally
			iPair := 0;
			status := SectionStatus.CLEARING;
			
		END_IF
		
	SectionStatus.CLEARING:
		ready := FALSE;
		busy := TRUE;
		done := FALSE;
	
		bundleOut := currentBundle;
		setConveyorMode(ConveyorMode.FORWARD);
		
		IF exitRefPos >= currentBundle.length AND NOT occupied THEN //rear of bundle has cleared the area
			status := SectionStatus.COMPLETE;
		END_IF
		
	SectionStatus.COMPLETE:	
		ready := FALSE;
		busy := FALSE;
		done := TRUE;
		
		iBundle := iBundle + 1;
		bundleOut := GVL.nullBundle;
		
		status := SectionStatus.IDLE;
		
	-100: //previously completed bundle reversed into this section
		ready := FALSE;
		busy := FALSE;
		done := done;
		
		IF NOT occupied THEN
			status := SectionStatus.ALIGNING;
		END_IF
		
END_CASE

PROPERTY PROTECTED accessConveyorMode : ConveyorMode
GET
accessConveyorMode := requestedConveyorMode;
END_GET
SET
requestedConveyorMode := accessConveyorMode;
END_SET
END_PROPERTY

PROPERTY accessNextSection : POINTER TO SectionEx
GET
accessNextSection := nextSection;
END_GET
SET
nextSection := accessNextSection;
END_SET
END_PROPERTY

PROPERTY PROTECTED accessPrevSection : POINTER TO SectionEx
GET
accessPrevSection := prevSection;
END_GET
SET
prevSection := accessPrevSection;
END_SET
END_PROPERTY

PROPERTY PROTECTED accessStatus : SectionStatus
GET
accessStatus := status;
END_GET
SET
status := accessStatus;
END_SET
END_PROPERTY

METHOD assignConveyors : BOOL
VAR_INPUT
	conveyorStart : INT;
	conveyorEnd : INT;
END_VAR
firstConveyor := conveyorStart;
lastConveyor := conveyorEnd;

assignConveyors := TRUE;
END_METHOD

METHOD ABSTRACT changeRobotsEOAT : BOOL
(*
IF robotLeft.tool <> sectionID THEN
	MEMSET(ADR(robotLeftOutputs), 0, SIZEOF(robotLeftOutputs));
	robotLeftOutputs[1] := A21.TOOL_CHANGE_CHIPBOARD;
	robotLeft.setParamsAndWait(robotLeftOutputs);
END_IF

IF robotRight.tool <> sectionID THEN
	MEMSET(ADR(robotRightOutputs), 0, SIZEOF(robotRightOutputs));
	robotRightOutputs[1] := A21.TOOL_CHANGE_CHIPBOARD;
	robotRight.setParamsAndWait(robotRightOutputs);
END_IF

changeRobotsEOAT := robotLeft.tool = sectionID AND robotRight.tool = sectionID;
*)
END_METHOD

METHOD connectTo : BOOL
VAR_INPUT
	connectedSection : POINTER TO SectionEx;
END_VAR
nextSection := connectedSection;
connectedSection^.prevSection := THIS;
END_METHOD

METHOD PROTECTED directionCheckAndSet : BOOL
VAR_INPUT
	conveyorRef : REAL;
	target : REAL;
END_VAR
//returns true conveyorRef is in range of target
IF InRange(conveyorRef - GVL.precisionTolerance, conveyorRef + GVL.precisionTolerance, target, EXCLUSIVE) THEN
	directionCheckAndSet := TRUE;
	
ELSIF conveyorRef > target THEN
	setConveyorMode(ConveyorMode.BACKWARD);
	
ELSIF conveyorRef < target THEN
	setConveyorMode(ConveyorMode.FORWARD);
	
END_IF
END_METHOD

METHOD PROTECTED discharge : BOOL
VAR_INPUT
END_VAR
END_METHOD

METHOD PROTECTED getConveyorMode : ConveyorMode;
getConveyorMode := requestedConveyorMode;
END_METHOD

METHOD getNext : POINTER TO SectionEx
VAR_INPUT
END_VAR
getNext := nextSection;
END_METHOD

METHOD ABSTRACT initHardware : BOOL
END_METHOD

METHOD PROTECTED ABSTRACT load : BOOL
VAR_INPUT
	pair : REFERENCE TO PositionMaterials;
END_VAR
(*
loading takes place while the section is NOT active
materials are loaded for the next incoming bundle, not the current bundle - may differ for each section
*)
END_METHOD

METHOD PROTECTED ABSTRACT process : BOOL
(*
VAR_INST
	iPair : USINT; //currentBundle.{material}[iPair]
	
	//case switches, iterators, counters
	step : INT := 0;
END_VAR
*)
(*
all material stations store a local conveyor encoder position (which may be negative)

conveyor operation is determined by all stations in order of priority - NTRL, FWD, BCK, STOP - refer to PackagerFreeAsync vars
stations request movement to place next material
stations stop the conveyor and operate on a bundle once the required position is reached

material slot loading is performed in the background on the fly
*)

//this method will likely be overriden by PaperEx
//UPDATE 2023-08-29 - this method is made abstract and will be implemented to each derived class


(*
CASE step OF
	0:
		IF place(iPair) THEN //finished placing and wrapping materials
			step := 10;
		END_IF
		
	10: //bundle finished, reset variables
		iPair := 0;
		step := 0;
		
		process := TRUE;
END_CASE
*)
END_METHOD

METHOD PROTECTED setConveyorMode : BOOL
VAR_INPUT
	newConveyorMode : ConveyorMode;
END_VAR
VAR
	prevSectionConveyorMode : ConveyorMode;
	
	i : INT;
END_VAR
requestedConveyorMode := newConveyorMode;

FOR i:=firstConveyor TO lastConveyor BY 1 DO
	
	CASE status OF
		SectionStatus.ALIGNING: //all conveyors request
			conveyors[i].setRequest(requestedConveyorMode);
			
		SectionStatus.ACTIVE, SectionStatus.CLEARING:
			//once previous bundle catches up, the conveyor that bundle sits on must be linked to this section
			//ConveyorControl() will take care of directional linking
			
			IF conveyors[i].occupied() THEN //follow this section's request
				conveyors[i].setRequest(requestedConveyorMode);
				
			ELSE //catch up succeeding bundle (FOLLOW PREVIOUS SECTION)
				IF prevSection <> 0 THEN
					conveyors[i].setRequest( prevSection^.getConveyorMode() );
				END_IF
			END_IF
	END_CASE	
	
END_FOR
END_METHOD

METHOD shiftIterator : BOOL
VAR
	i : INT;
END_VAR
//2023-10-24 - array of pointers replaced with iterator for MAIN's queue passed by pointer
iBundle := iBundle - 1;
END_METHOD

METHOD PROTECTED ABSTRACT usesProcess : BOOL
END_METHOD

END_FUNCTION_BLOCK

// ---- Sections/Concrete/CardboardCornerGuardEx.TcPOU
FUNCTION_BLOCK CardboardCornerGuardEx EXTENDS SectionEx
VAR
	robotLeft, robotRight : REFERENCE TO Robot;
	
	insertionLeft, insertionRight : REFERENCE TO Insertion;
	insertionBottom : REFERENCE TO TeknicEIP;
	
	wrapper : REFERENCE TO WrapMachine;
	overhead : REFERENCE TO STRING;
	
	skidLeft, skidRight : REFERENCE TO MaterialStorage; //cardboard
	magazineLeft, magazineRight : REFERENCE TO MaterialStorage; //corner guard
	
	benderLeft : REFERENCE TO FoldingMachine;
END_VAR
VAR
	pushConveyorPos: REAL;
	wrapConveyorPos : REAL;
	
	insertionSlots : ARRAY[Surface.TOP_LEFT..Surface.BOTTOM_RIGHT] OF STRING;
	
	combinedCardboardCornerGuard : ARRAY[0..2*GVL.maxPairs] OF PositionMaterials;
	recipesCombined : BOOL;
	
	materialsArr : POINTER TO PositionMaterials; //array of PositionMaterials
	currentPair : REFERENCE TO PositionMaterials;
	
	frontCoverPlaced : BOOL;
	backCoverPlaced : BOOL;
	
	cornerSetLeft, cornerSetRight : INT;
	
	iWrap : INT;
	
	step : (PLACE_FRONT_COVER := -10, PLACE_BACK_COVER := -20, RUN_TO_POSITION, LOAD_FLATS, PUSH, RUN_TO_WRAP_POSITION, WRAP_AND_RELEASE, RESET);
	robotLeftOutputs, robotRightOutputs : ARRAY[1..50] OF INT;
END_VAR

entryRefPos := pushConveyorPos;
exitRefPos := wrapConveyorPos;

SUPER^();

CASE status OF
	SectionStatus.IDLE:
		RETURN;
	
	SectionStatus.ALIGNING:
		IF NOT recipesCombined THEN
			combine(
				currentBundle.cardboard, 
				currentBundle.cornerGuard, 
				combinedCardboardCornerGuard, 
				currentBundle.cardboard_over_cornerGuard);
				
			recipesCombined := TRUE;
		END_IF
		
	SectionStatus.ACTIVE:
		recipesCombined := FALSE;
		
	SectionStatus.CLEARING:
		//
		
	SectionStatus.COMPLETE:	
		//
		
	-100:
		RETURN;
		
END_CASE

METHOD changeRobotsEOAT : BOOL
VAR_INPUT
END_VAR
(*
IF robotLeft.tool <> sectionID THEN
	MEMSET(ADR(robotLeftOutputs), 0, SIZEOF(robotLeftOutputs));
	//robotLeftOutputs[1] := A21.TOOL_CHANGE_CHIPBOARD;
	robotLeft.setParamsAndWait(robotLeftOutputs);
END_IF

IF robotRight.tool <> sectionID THEN
	MEMSET(ADR(robotRightOutputs), 0, SIZEOF(robotRightOutputs));
	//robotRightOutputs[1] := A21.TOOL_CHANGE_CHIPBOARD;
	robotRight.setParamsAndWait(robotRightOutputs);
END_IF

changeRobotsEOAT := robotLeft.tool = sectionID AND robotRight.tool = sectionID;
*)
END_METHOD

METHOD PROTECTED combine : BOOL
VAR_IN_OUT
	cardboard : ARRAY[*] OF PositionMaterials;
	cornerGuard : ARRAY[*] OF PositionMaterials;
	
	combined : ARRAY[*] OF PositionMaterials;
END_VAR
VAR_INPUT
	cardboard_over_cornerGuard : BOOL;
END_VAR
VAR_INST
	topLength : REAL;
	leftLength : REAL;
	rightLength : REAL;
	bottomLength : REAL;
	
	topLeftLength : REAL;
	topRightLength : REAL;
	bottomLeftLength : REAL;
	bottomRightLength : REAL;
	
	outerMaterialLength : REAL;
	innerMaterialLength : REAL;
	
	i : INT;
	iCardboard : INT;
	iCornerGuard : INT;
END_VAR
FOR i:=0 TO GVL.maxPairs*2 BY 1 DO
	IF //no more cardboard (reached end of array or unused entries), 
		(iCardboard >= GVL.maxPairs OR_ELSE NOT PositionIsValid(cardboard[iCardboard])) AND_THEN //no more valid cardboard entries
		iCornerGuard < GVL.maxPairs AND_THEN //still has remaining corner guard
		PositionIsValid(cornerGuard[iCornerGuard]) //remaining corner guard is valid		
	THEN //finish with cornerguard
		combined[i] := cornerGuard[iCornerGuard];
		iCornerGuard := iCornerGuard + 1;
		CONTINUE;
	END_IF
	
	IF //no more cornerguard (reached end of array or unused entries)
		(iCornerGuard >= GVL.maxPairs OR_ELSE NOT PositionIsValid(cornerGuard[iCornerGuard])) AND_THEN
		iCardboard < GVL.maxPairs AND_THEN
		PositionIsValid(cardboard[iCardboard])
	THEN //finish with cardboard
		combined[i] := cardboard[iCardboard];
		iCardboard := iCardboard + 1;
		CONTINUE;
	END_IF
	
	(*
	IF NOT cardboard_over_cornerGuard THEN //cardboard on inside
		setOrder(cardboard, cornerGuard, combined, iCardboard, iCornerGuard, i);
		
	ELSE //cardboard on outside
		setOrder(cornerGuard, cardboard, combined, iCornerGuard, iCardboard, i);
		
	END_IF
	*)
END_FOR

combine := TRUE;
END_METHOD

METHOD initHardware : BOOL
conveyors := ADR(allConveyors);

robotLeft REF= robots[3];
robotRight REF= robots[4];
(*
insertionLeft REF= Hardware.insertionCardboardCornerGuardSides[Surface.LEFT];
insertionRight REF= Hardware.insertionCardboardCornerGuardSides[Surface.RIGHT];

wrapper REF= Hardware.wrapperCardboardCornerguard;
overhead REF= Hardware.overhead;

skidLeft REF= Hardware.cardboardSkid[Surface.LEFT];
skidRight REF= Hardware.cardboardSkid[Surface.RIGHT];

magazineLeft REF= Hardware.cornerGuardMagazine[Surface.LEFT];
magazineRight REF= Hardware.cornerGuardMagazine[Surface.RIGHT];

benderLeft REF= Hardware.cardboardBender[Surface.LEFT];
*)

insertionLeft REF= insertionA22Left;
insertionRight REF= insertionA22Right;

wrapper REF= wrapperA22;
overhead REF= Hardware.overhead;

skidLeft REF= cardboardSkidLeft;
skidRight REF= cardboardSkidRight;

magazineLeft REF= cornerGuardMagazineLeft;
magazineRight REF= cornerGuardMagazineRight;

benderLeft REF= cardboardBenderLeft;
END_METHOD

METHOD PROTECTED leftBendingSequence : BOOL
VAR_IN_OUT
	actingRobot : Robot;
	actingSkid : MaterialStorage;
	
	actingLoadStep : INT;
	actingRobotStep : INT;
END_VAR
VAR_INPUT
	materialID : STRING;
	foldPosition1 : INT;
	foldPosition2 : INT;
END_VAR
VAR_OUTPUT
	fail : BOOL;
END_VAR
VAR
	slot : INT;
END_VAR
END_METHOD

METHOD PROTECTED leftOverheadSequence : BOOL
VAR_IN_OUT
	actingRobot : Robot;
	actingSkid : MaterialStorage;
	
	actingLoadStep : INT;
	actingRobotStep : INT;
END_VAR
VAR_INPUT
	materialID : STRING;
	foldPosition1 : INT;
	foldPosition2 : INT;
END_VAR
VAR_OUTPUT
	fail : BOOL;
END_VAR
VAR
	slot : INT;
END_VAR
(*
CASE actingLoadStep OF
	0: //skid to bender
		IF NOT actingSkid.findSlot(materialID, position=> slot) THEN
			fail := TRUE;
			RETURN;
		END_IF
		
		IF
			actingRobot.reserve() AND_THEN
			actingRobot.setCommandAndWait(
				task:= A22.TRANSFER_TO_BENDER, 
				param0:= slot, 
				param1:= foldPosition1, 
				param2:= foldPosition2)
		THEN
			actingRobotStep := 10;
		END_IF
		
	10: //bend
		(*
		IF bendingMachine.done THEN
			cardboardCornersLoadStep := 20;
		END_IF
		*)
		
	20: //bender to overhead
		IF overhead <> '' THEN
			RETURN;
		END_IF
		
		IF
			actingRobot.reserve() AND_THEN
			actingRobot.setCommandAndWait(
				task:= A22.TRANSFER_TO_OVERHEAD, 
				param0:= 0, 
				param1:= 0, 
				param2:= 0)
		THEN
			actingRobotStep := 10;
		END_IF
		
		CASE actingRobotStep OF
			COMMAND: //send command
				IF NOT actingRobot.reserve() THEN
					RETURN;
				END_IF
				
				IF actingSkid.findSlot(currentPair.topRight, position=> slot) THEN
					actingRobot.command(
						task:= A22.TRANSFER_TO_OVERHEAD, 
						param0:= 0, 
						param1:= 0, 
						param2:= 0);
						
				ELSE
					fail := TRUE;
					RETURN;
					
				END_IF
				
			WAIT:
				IF actingRobot.done THEN
					overhead := materialID;
					
					actingRobot.release();
					actingRobotStep := 30;
					actingLoadStep := Surface.BOTTOM_RIGHT;
				END_IF
		END_CASE
END_CASE
*)
END_METHOD

METHOD PROTECTED leftRobotCornersSequence : BOOL
VAR_IN_OUT
	actingRobot : Robot;
	skid : MaterialStorage;
	loadStep : INT;
END_VAR
VAR_INPUT
	surfaceID : Surface;
	materialID : STRING;
	foldPos0 : INT;
	foldPos1 : INT;
END_VAR
VAR_OUTPUT
	fail : BOOL;
END_VAR
VAR
	slot : INT;
	
	task : INT;
	param0, param1, param2 : INT;
END_VAR
IF materialID = '' THEN
	leftRobotCornersSequence := TRUE;
	RETURN;
END_IF

IF NOT benderLeft.busy THEN
	benderLeft.foldPos0 := foldPos0;
	benderLeft.foldPos1 := foldPos1;
END_IF

CASE loadStep OF
	0: //skid to bender
		IF NOT skid.findSlot(materialID, atSlot=> slot) THEN
			fail := TRUE;
			RETURN;
		END_IF
		
		IF
			actingRobot.setCommandAndWait(
				task:= A22.TRANSFER_TO_BENDER, 
				param1:= slot, 
				param2:= foldPos0, 
				param3:= foldPos1)
		THEN
			loadStep := 10;
		END_IF
		
	10: //bend
		//IF benderLeft.done THEN
			loadStep := 20;
		//END_IF
		
		
	20: //bender to overhead or left insertion
		CASE surfaceID OF
			Surface.TOP_RIGHT, Surface.BOTTOM_RIGHT: //transfer to overhead
				IF overhead <> '' THEN
					RETURN;
				END_IF
				task := A22.TRANSFER_TO_OVERHEAD;
				
			Surface.TOP_LEFT: //load to insertion
				task:= A22.LOAD_BENDER_TO_UPPER_CORNER;
					
			Surface.BOTTOM_LEFT: //load to insertion
				task := A22.LOAD_BENDER_TO_LOWER_CORNER;
				
		END_CASE
		
		IF
			actingRobot.setCommandAndWait(
				task:= task, 
				param1:= param0, 
				param2:= param1, 
				param3:= param1)
		THEN
			 loadStep := COMPLETE;
		END_IF
	
	COMPLETE:
		//turn on suction
		leftRobotCornersSequence := TRUE;
	
END_CASE
END_METHOD

METHOD PROTECTED load : BOOL
VAR_INPUT
	pair : REFERENCE TO PositionMaterials;
END_VAR
VAR
	nextPair : REFERENCE TO PositionMaterials REF= materialsArr[iPair + 1];
	finished : BOOL;
END_VAR
(*
this method only loads corner materials (L-cardboards and corner guards)
to load flat cardboards, use loadFlats()
*)

IF NOT (robotLeft.operational AND robotRight.operational) THEN
	error := TRUE;
	currentBypass := TRUE;
	RETURN;
END_IF

IF NOT (robotLeft.reserve(sectionID) AND robotRight.reserve(sectionID)) THEN //both robots must be reserved first
	RETURN;
END_IF


IF //if next material has same position as this material, only happens if this material is cardboard and next is corner guard
	nextPair.position = pair.position AND_THEN
	NOT loadCornerGuards(nextPair, fail=> ) //load next pair (corner guards) first
THEN
	RETURN;
END_IF


IF MatchesMaterialType(pair:= pair, materialType:= 'CAR') THEN //is cardboard
	load := loadCornerCardboards(pair:= pair);

ELSIF MatchesMaterialType(pair:= pair, materialType:= 'COR') THEN //is corner guard
	load := loadCornerGuards(pair:= pair);

END_IF


IF load THEN
	robotLeft.release(sectionID);
	robotRight.release(sectionID);
END_IF
END_METHOD

METHOD PROTECTED loadBottom : BOOL
VAR_IN_OUT
	actingRobot : Robot;
	actingStorage : MaterialStorage;
	actingLoadStep : INT;
END_VAR
VAR_INPUT
	material : STRING;
END_VAR
VAR_OUTPUT
	fail : BOOL;
END_VAR
VAR
	slot : INT;
END_VAR
IF material = '' THEN
	loadBottom := TRUE;
	RETURN;
END_IF

CASE actingLoadStep OF
	0:
		IF NOT actingStorage.findSlot(materialID := material, atSlot => slot) THEN
			fail := TRUE;
			RETURN;
		END_IF
		
		IF
			actingRobot.setCommandAndWait( //perform the task
				task:= A22.LOAD_CARDBOARD_BOTTOM,
				param1:= slot,
				param2:= 0,
				param3:= 0)
		THEN
			actingLoadStep := COMPLETE;
		END_IF
		
	COMPLETE:
		//turn on suction
		loadBottom := TRUE;
	
END_CASE
END_METHOD

METHOD PROTECTED loadBottomLeft : BOOL
VAR_IN_OUT
	actingRobot : Robot;
	actingStorage : MaterialStorage;
	actingLoadStep : INT;
END_VAR
VAR_INPUT
	material : STRING;
END_VAR
VAR_OUTPUT
	fail : BOOL;
END_VAR
VAR
	slot : INT;
END_VAR
IF material = '' THEN
	loadBottomLeft := TRUE;
	RETURN;
END_IF

